# B&R Automation Studio project NAEUL004C00R13L518F00 (part 37)

### NtParam.typ - Change By Project
```iecst
(*2020-07-28*)

TYPE
	eNtParamAction :
		(
		NtParamActIdle,
		NtParamActCreateDir,
		NtParamActRead,
		NtParamActWrite,
		NtParamActLoad,
		NtParamActSave
		);
	tyNtParam : 	STRUCT
		tyDISettings : tyDigitalInputSettings := (diSafetyRlySig:=1,diEStopSig:=2,diCoverSWSig:=3,diUBAA:=4,diUBAB:=5,diUBAAStat:=6,diUBABStat:=7,diPusherExtRS:=12,diPusherRetRS:=13,diConvLftSen:=27,diConvMidSen:=28,diConvRgtSen:=29,diConvClrSen:=30,diOvenInfeedSigA:=0,diOvenInfeedSigB:=0,diLifterTimingBeltSen:=10,diLifterSafetyLmtSW1:=11,diLifterSafetyLmtSW2:=0,diMag1FixedClampRS:=0,diMag1FixedUnclampRS:=0,diMag1RemoteClampRS:=0,diMag1RemoteUnclampRS:=0,diMag2FixedClampRS:=0,diMag2FixedUnclampRS:=0,diMag2RemoteClampRS:=0,diMag2RemoteUnclampRS:=0,diMag3FixedClampRS:=0,diMag3FixedUnclampRS:=0,diMag3RemoteClampRS:=0,diMag3RemoteUnclampRS:=0,diInShutterOpenRS:=14,diInShutterCloseRS:=15,diOutShutterOpenRS:=16,diOutShutterCloseRS:=17,diMagPresentSen1:=8,diMagPresentSen2:=9,diMagPresentSen3:=0,diMagConvEntSen1:=0,diMagConvEntSen2:=0,diMagConvEntSen3:=0,diMag1AIVInPosSen1:=0,diMag1AIVInPosSen2:=0,diMag2AIVInPosSen1:=0,diMag2AIVInPosSen2:=0,diMag3AIVInPosSen1:=0,diMag3AIVInPosSen2:=0,diMag1OrientChkSen1:=0,diMag1OrientChkSen2:=0,diMag2OrientChkSen1:=0,diMag2OrientChkSen2:=0,diMag3OrientChkSen1:=0,diMag3OrientChkSen2:=0,diUSWidthChkSen:=0,diConvLineAInletSen:=0,diConvLineBInletSen:=0,diMagConvHeightSen1:=0,diMagConvHeightSen2:=0,diMagConvHeightSen3:=0,diMagConvSmallMagSen1:=0,diMagConvSmallMagSen2:=0,diMagConvSmallMagSen3:=0,diMagConvLargeMagSen1:=0,diMagConvLargeMagSen2:=0,diMagConvLargeMagSen3:=0,diMagConvCAB717MagSen1:=0,diMagConvCAB717MagSen2:=0,diMagConvCAB717MagSen3:=0,diMag1SelUnClampRS:=0,diMag2SelUnClampRS:=0,diMag3SelUnClampRS:=0,diMag1WallEngageRS:=0,diMag1WallDisengageRS:=0,diMag2WallEngageRS:=0,diMag2WallDisengageRS:=0,diMag3WallEngageRS:=0,diMag3WallDisengageRS:=0,diMag1SafetyBarExtRS:=0,diMag1SafetyBarRetRS:=0,diMag2SafetyBarExtRS:=0,diMag2SafetyBarRetRS:=0,diMag3SafetyBarExtRS:=0,diMag3SafetyBarRetRS:=0,diSOT1Receive:=0,diSOT1AIVError:=0,diSOT1AIVSizeLarge:=0,diSOT1AIVReady:=0,diSOT1AIVAvailable:=0,diSOT2Receive:=0,diSOT2AIVError:=0,diSOT2AIVSizeLarge:=0,diSOT2AIVReady:=0,diSOT2AIVAvailable:=0,diSOT3Receive:=0,diSOT3AIVError:=0,diSOT3AIVSizeLarge:=0,diSOT3AIVReady:=0,diSOT3AIVAvailable:=0,diSOT4Receive:=0,diSOT4AIVError:=0,diSOT4AIVSizeLarge:=0,diSOT4AIVReady:=0,diSOT4AIVAvailable:=0,diFleetManagerReady:=0,diPusherExtSlwSen:=0,diPusherRetSlwSen:=0,diMtrPshrTorqueSig:=0,diMtrPshrAlmSig:=0,diMagWidthChkSen:=0,diPshrAntiJam:=0,diInMagConvEntSen:=0,diInMagConvExtSen:=0,diInMagConvMidSen:=0,diOutMagConvEntSen:=0,diOutMagConvExtSen:=0,diOutMagConvMidSen:=0,diInMagConv2EntSen:=0,diInMagConv2ExtSen:=0,diInMagConv2MidSen:=0,diOutMagConv2EntSen:=0,diOutMagConv2ExtSen:=0,diOutMagConv2MidSen:=0,diLifterLmtSW:=0,diLifter2LmtSW:=0,diMtrOverloadSig:=0,diOutShutterOpenRS2:=0,diOutShutterCloseRS2:=0,diOutShutterOpenRS3:=0,diOutShutterCloseRS3:=0,diMag1FixedClampSen:=0,diMag2FixedClampSen:=0,diMag3FixedClampSen:=0,diCurtainSenPB:=0,diCurtainSen:=0,diCurtainSafetySig:=0,diHighMagDetSen1:=0,diHighMagDetSen2:=0,diHighMagDetSen3:=0,diInletStopperASen:=0,diScanComplSig:=0,diPCBScanSen:=0,diSPARE17:=0,diSPARE18:=0,diSPARE19:=0,diSPARE20:=0);
		tyDOSettings : tyDigitalOutputSettings := (diSafetyRlyRst:=1,diTLRed:=4,diTLAmber:=3,diTLGreen:=2,diBuzzer:=5,diUSBA:=8,diUSBB:=9,diOvenInfoSigA:=7,diOvenInfoSigB:=10,diPusherExtCtrl:=11,diStopperUnblkCtrlA:=0,diStopperUnblkCtrlB:=0,diMag1FixedClampCtrl:=0,diMag1RemoteClampCtrl:=0,diMag2FixedClampCtrl:=0,diMag2RemoteClampCtrl:=0,diMag3FixedClampCtrl:=0,diMag3RemoteClampCtrl:=0,diInShutterOpenCtrl:=15,diInShutterCloseCtrl:=16,diOutShutterOpenCtrl:=17,diOutShutterCloseCtrl:=18,diMag1ConvMtrIn:=0,diMag1ConvMtrOut:=0,diMag2ConvMtrIn:=0,diMag2ConvMtrOut:=0,diMag3ConvMtrIn:=0,diMag3ConvMtrOut:=0,diMag1SelClampCtrl:=0,diMag2SelClampCtrl:=0,diMag3SelClampCtrl:=0,diPushConvMtrOn:=12,diMag1WallEngageCtrl:=0,diMag2WallEngageCtrl:=0,diMag3WallEngageCtrl:=0,diMag1SafetyBarRetCtrl:=0,diMag2SafetyBarRetCtrl:=0,diMag3SafetyBarRetCtrl:=0,diSOT1MagError:=0,diSOT1MagSizeLarge:=0,diSOT1MagReady:=0,diSOT1MagAvailable:=0,diSOT2MagError:=0,diSOT2MagSizeLarge:=0,diSOT2MagReady:=0,diSOT2MagAvailable:=0,diSOT3MagError:=0,diSOT3MagSizeLarge:=0,diSOT3MagReady:=0,diSOT3MagAvailable:=0,diSOT4MagError:=0,diSOT4MagSizeLarge:=0,diSOT4MagReady:=0,diSOT4MagAvailable:=0,diMagAWOpenLimByp1:=0,diMagAWOpenLimByp2:=0,diMagAWOpenLimByp3:=0,diMagAWOpenLimByp4:=0,diMagAWSmallLimSen1:=0,diMagAWSmallLimSen2:=0,diMagAWSmallLimSen3:=0,diMagAWSmallLimSen4:=0,diMag1ReqToBring:=0,diMag1ReqToGet:=0,diMag2ReqToBring:=0,diMag2ReqToGet:=0,diMag3ReqToBring:=0,diMag3ReqToGet:=0,diMag4ReqToBring:=0,diMag4ReqToGet:=0,diMtrPshrExt:=0,diMtrPshrRet:=0,diMtrPshrOn:=0,diMtrPshrBrakeRls:=0,diMtrPshrSpdBinBit0:=0,diMtrPshrSpdBinBit1:=0,diMtrPshrSpdBinBit2:=0,diMtrPshrAlmRst:=0,diInMagConvMtrOn:=0,diOutMagConvMtrOn:=0,diInMagConv2MtrOn:=0,diOutMagConv2MtrOn:=0,diEntTopStprUnblkCtrl:=0,diMidTopStprUnblkCtrl:=0,diExtTopStprUnblkCtrl:=0,diMidBtmStprUnblkCtrl:=0,diExtBtmStprUnblkCtrl:=0,diEntTopStprUnblkCtrl2:=0,diMidTopStprUnblkCtrl2:=0,diExtTopStprUnblkCtrl2:=0,diMidBtmStprUnblkCtrl2:=0,diExtBtmStprUnblkCtrl2:=0,diMtrPwrRly:=0,diMag1FixedClampOpenCtrl:=0,diMag1RemoteClampOpenCtrl:=0,diMag2FixedClampOpenCtrl:=0,diMag2RemoteClampOpenCtrl:=0,diMag3FixedClampOpenCtrl:=0,diMag3RemoteClampOpenCtrl:=0,diOutShutterOpenCtrl2:=0,diOutShutterCloseCtrl2:=0,diOutShutterOpenCtrl3:=0,diOutShutterCloseCtrl3:=0,diBypCurtainSen:=0,diRstCurtainSen:=0,diBypCurtainPBLED:=6,diInletStopperRetCtrl:=0,diInletStopperExtCtrl:=0,diScanTrigSig:=0,diMag1ExitPCB:=0,diMag2ExitPCB:=0,diMag3ExitPCB:=0,diMag1SelUnClampCtrl:=0);
		bAWPusherPrep : BOOL := FALSE;
		bAWPrep : BOOL := TRUE;
		bLFPrep : BOOL := TRUE;
		bLeaderMc : BOOL := FALSE;
		bLFUsrSetPrep : BOOL := TRUE;
		diLFWidthLimit : DINT := 3000;
		bLFProdWidthChk : BOOL := FALSE;
		bUSWidthChkPrep : BOOL := FALSE;
		bLCSLFPrep : BOOL := TRUE;
		bLCSReqRcpPrep : BOOL := TRUE;
		bLCSManageRcpPrep : BOOL := TRUE;
		bLCSLiveDatPrep : BOOL := TRUE;
		bIPCSMEMA9851ExtdPrep : BOOL := TRUE;
		bVSMEMAPrep : BOOL := TRUE;
		bHermesPrep : BOOL := FALSE;
		bHermesRmtPrep : BOOL := FALSE;
		bOvenInfoPrep : BOOL := TRUE;
		bOvenInfoExtdPrep : BOOL := FALSE;
		bSSaverPrep : BOOL := TRUE;
		diAWPushPulOffsetInUM : DINT := 0;
		diWidthOffsetInUM : DINT := 0;
		sJobNo : STRING[30] := '2023-0529E01';
		usiNtAddr : USINT := 4;
		bProjLifterMagPlatform : BOOL := TRUE;
		bProjLaneBPrep : BOOL := FALSE;
		bProjBrdPerSltPrep : BOOL := FALSE;
		bProjLongBrdPrep : BOOL := FALSE;
		bProjInletShutPrep : BOOL := TRUE;
		bProjOutletShutPrep : BOOL := TRUE;
		bProjStopperAPrep : BOOL := FALSE;
		bProjStopperBPrep : BOOL := FALSE;
		bProjMag1ConvPrep : BOOL := FALSE;
		bProjMag2ConvPrep : BOOL := FALSE;
		bProjMag3ConvPrep : BOOL := FALSE;
		bProjLifter2Prep : BOOL := FALSE;
		bProjMagConvLane1Prep : BOOL := FALSE; (*TopBtm Conv, Lifter Conv*)
		bProjMagConvLane2Prep : BOOL := FALSE; (*TopBtm Conv, Lifter Conv*)
		bProjTopEntStprPrep : BOOL := FALSE; (*TopBtm Conv, Lifter Conv*)
		bProjTopMidStprPrep : BOOL := FALSE; (*TopBtm Conv, Lifter Conv*)
		bProjTopExtStprPrep : BOOL := FALSE; (*TopBtm Conv, Lifter Conv*)
		bProjBtmMidStprPrep : BOOL := FALSE; (*TopBtm Conv, Lifter Conv*)
		bProjBtmExtStprPrep : BOOL := FALSE; (*TopBtm Conv, Lifter Conv*)
		bProjTopEntStprPrep2 : BOOL := FALSE; (*TopBtm Conv, Lifter Conv*)
		bProjTopMidStprPrep2 : BOOL := FALSE; (*TopBtm Conv, Lifter Conv*)
		bProjTopExtStprPrep2 : BOOL := FALSE; (*TopBtm Conv, Lifter Conv*)
		bProjBtmMidStprPrep2 : BOOL := FALSE; (*TopBtm Conv, Lifter Conv*)
		bProjBtmExtStprPrep2 : BOOL := FALSE; (*TopBtm Conv, Lifter Conv*)
		bProjMagOrientChkSenPrep : BOOL := FALSE;
		bProjAGVPrep : BOOL := FALSE;
		bProjTCPAGVSigPrep : BOOL := FALSE;
		bProjBypsInitConvPrep : BOOL := TRUE;
		bProjRlsNewProdPrep : BOOL := FALSE;
		bProjBtnInsertRmvMag : BOOL := TRUE; (*fixed type*)
		bProjSOTSensorPrep : BOOL := FALSE;
		bProjMotorizedPusherPrep : BOOL := FALSE;
		bProjMagAWPrep : BOOL := FALSE;
		bProjMagSafetyBarPrep : BOOL := TRUE;
		diProjMagMinSlt : DINT := 1;
		diProjMagMaxSlt : DINT := 50;
		eProjMag : eULMag := ULMagTriple;
		eProjConvDir : eConvDir := ConvDirLToR;
		eProjMagConvDir : eConvDir := ConvDirLToL;
		eProjMagBuffferActLoad : eLifMagULUpdateData := BufferActLoadWhenStarted;
		eProjInMagConvDir : eConvDir := ConvDirRToL; (*Top*)
		eProjOutMagConvDir : eConvDir := ConvDirLToR; (*Bottom*)
		eProjLifterMagConvDir : eConvDir := ConvDirRToR; (*LifterConv*)
		eProjInMagConv2Dir : eConvDir := ConvDirRToL; (*Top*)
		eProjOutMagConv2Dir : eConvDir := ConvDirLToR; (*Bottom*)
		eProjLifterMagConv2Dir : eConvDir := ConvDirRToR; (*LifterConv*)
		sUsrFolderProgNm : STRING[15] := 'UsrFolder';
		sLibVersionProgNm : STRING[15] := 'LibVer';
		sTimeProgNm : STRING[15] := 'Time';
		sHWInfoProgNm : STRING[15] := 'HWInfo';
		sHWInfoDevice : STRING[3] := 'IF2';
		tyTLBuz : tyTLBuzIn1;
		sAlmProgNm : STRING[15] := 'Alarm';
		udiAlmFileKeepDay : UDINT := 30;
		sProdRcpProgNm : STRING[15] := 'ProdRcp';
		sProdRcpListFileNm : STRING[80] := 'ProductRecipeList.dat';
		sProdRcpSingleFileNm : STRING[80] := 'ProductRecipe.dat';
		sMpProdRcpProgNm : STRING[15] := 'MpProdRcp';
		sMpProdRcpFileNm : STRING[255] := 'MpProductRecipe.xml';
		sMpProdRcpPVNm : STRING[100] := 'MpProdRcp:a_tyMpProdRcp1';
		sMagRcpProgNm : STRING[15] := 'MagRcp';
		sMagRcpListFileNm : STRING[80] := 'MagazineRecipeList.dat';
		sMagRcpSingleFileNm : STRING[80] := 'MagazineRecipe.dat';
		sMcParamProgNm : STRING[15] := 'McParam';
		sMcParamFileNm : STRING[80] := 'MachineParameter.dat';
		sUsrMgmtProgNm : STRING[15] := 'UsrMgmt';
		sBffr1ProgNm : STRING[15] := 'Buffer 1';
		sBffr1FileNm : STRING[80] := 'Buffer1.dat';
		bBffr1NxtLoadSeq : BOOL := TRUE;
		sBffr2ProgNm : STRING[15] := 'Buffer 2';
		sBffr2FileNm : STRING[80] := 'Buffer2.dat';
		bBffr2NxtLoadSeq : BOOL := TRUE;
		sBffr3ProgNm : STRING[15] := 'Buffer 3';
		sBffr3FileNm : STRING[80] := 'Buffer3.dat';
		bBffr3NxtLoadSeq : BOOL := TRUE;
		sUSSMEMAAProgNm : STRING[15] := 'USSMEMA A';
		tUSSMEMAARstDlyTm : TIME := T#500ms;
		tUSSMEMAASigInChkTm : TIME := T#100ms;
		sUSSMEMABProgNm : STRING[15] := 'USSMEMA B';
		tUSSMEMABRstDlyTm : TIME := T#500ms;
		tUSSMEMABSigInChkTm : TIME := T#100ms;
		sUSSMEMA1ProgNm : STRING[15] := 'Mag1_US';
		tUSSMEMA1RstDlyTm : TIME := T#0s;
		tUSSMEMA1SigInChkTm : TIME := T#100ms;
		sUSSMEMA2ProgNm : STRING[15] := 'Mag2_US';
		tUSSMEMA2RstDlyTm : TIME := T#0s;
		tUSSMEMA2SigInChkTm : TIME := T#100ms;
		sUSSMEMA3ProgNm : STRING[15] := 'Mag3_US';
		tUSSMEMA3RstDlyTm : TIME := T#0s;
		tUSSMEMA3SigInChkTm : TIME := T#100ms;
		sDSSMEMA1ProgNm : STRING[15] := 'Mag1_DS';
		tDSSMEMA1RstDlyTm : TIME := T#0s;
		tDSSMEMA1SigInChkTm : TIME := T#100ms;
		sDSSMEMA2ProgNm : STRING[15] := 'Mag2_DS';
		tDSSMEMA2RstDlyTm : TIME := T#0s;
		tDSSMEMA2SigInChkTm : TIME := T#100ms;
		sDSSMEMA3ProgNm : STRING[15] := 'Mag3_DS';
		tDSSMEMA3RstDlyTm : TIME := T#0s;
		tDSSMEMA3SigInChkTm : TIME := T#100ms;
		sInShutterProgNm : STRING[15] := 'Inlet Shutter';
		bInShutterTwoCtrlIn : BOOL := TRUE;
		tInShutterExtTO : TIME := T#20s;
		tInShutterRetTO : TIME := T#20s;
		sOutShutterProgNm : STRING[15] := 'Outlet Shutter';
		bOutShutterTwoCtrlIn : BOOL := TRUE;
		tOutShutterExtTO : TIME := T#20s;
		tOutShutterRetTO : TIME := T#20s;
		sSelClamp1ProgNm : STRING[15] := 'Sel Clamp 1';
		bSelClamp1TwoCtrlIn : BOOL := TRUE;
		tSelClamp1ExtDlyTm : TIME := T#10s;
		tSelClamp1RetDlyTm : TIME := T#10s;
		sSelClamp2ProgNm : STRING[15] := 'Sel Clamp 2';
		bSelClamp2TwoCtrlIn : BOOL := FALSE;
		tSelClamp2ExtDlyTm : TIME := T#10s;
		tSelClamp2RetDlyTm : TIME := T#10s;
		sSelClamp3ProgNm : STRING[15] := 'Sel Clamp 3';
		bSelClamp3TwoCtrlIn : BOOL := FALSE;
		tSelClamp3ExtDlyTm : TIME := T#10s;
		tSelClamp3RetDlyTm : TIME := T#10s;
		sTopEntStprProgNm : STRING[15] := 'Top Ent Stpr';
		bTopEntStprTwoCtrlIn : BOOL := FALSE;
		tTopEntStprExtDlyTm : TIME := T#1s;
		tTopEntStprRetDlyTm : TIME := T#1s;
		sTopMidStprProgNm : STRING[15] := 'Top Mid Stpr';
		bTopMidStprTwoCtrlIn : BOOL := FALSE;
		tTopMidStprExtDlyTm : TIME := T#1s;
		tTopMidStprRetDlyTm : TIME := T#1s;
		sTopExtStprProgNm : STRING[15] := 'Top Ext Stpr';
		bTopExtStprTwoCtrlIn : BOOL := FALSE;
		tTopExtStprExtDlyTm : TIME := T#1s;
		tTopExtStprRetDlyTm : TIME := T#1s;
		sBtmMidStprProgNm : STRING[15] := 'Top Mid Stpr';
		bBtmMidStprTwoCtrlIn : BOOL := FALSE;
		tBtmMidStprExtDlyTm : TIME := T#1s;
		tBtmMidStprRetDlyTm : TIME := T#1s;
		sBtmExtStprProgNm : STRING[15] := 'Btm Ext Stpr';
		bBtmExtStprTwoCtrlIn : BOOL := FALSE;
		tBtmExtStprExtDlyTm : TIME := T#1s;
		tBtmExtStprRetDlyTm : TIME := T#1s;
		sTopEntStprProgNm2 : STRING[15] := 'Top Ent Stpr2';
		bTopEntStprTwoCtrlIn2 : BOOL := FALSE;
		tTopEntStprExtDlyTm2 : TIME := T#1s;
		tTopEntStprRetDlyTm2 : TIME := T#1s;
		sTopMidStprProgNm2 : STRING[15] := 'Top Mid Stpr2';
		bTopMidStprTwoCtrlIn2 : BOOL := FALSE;
		tTopMidStprExtDlyTm2 : TIME := T#1s;
		tTopMidStprRetDlyTm2 : TIME := T#1s;
		sTopExtStprProgNm2 : STRING[15] := 'Top Ext Stpr2';
		bTopExtStprTwoCtrlIn2 : BOOL := FALSE;
		tTopExtStprExtDlyTm2 : TIME := T#1s;
		tTopExtStprRetDlyTm2 : TIME := T#1s;
		sBtmMidStprProgNm2 : STRING[15] := 'Top Mid Stpr2';
		bBtmMidStprTwoCtrlIn2 : BOOL := FALSE;
		tBtmMidStprExtDlyTm2 : TIME := T#1s;
		tBtmMidStprRetDlyTm2 : TIME := T#1s;
		sBtmExtStprProgNm2 : STRING[15] := 'Btm Ext Stpr2';
		bBtmExtStprTwoCtrlIn2 : BOOL := FALSE;
		tBtmExtStprExtDlyTm2 : TIME := T#1s;
		tBtmExtStprRetDlyTm2 : TIME := T#1s;
		sStopperAProgNm : STRING[15] := 'Stopper A';
		bStopperATwoCtrlIn : BOOL := FALSE;
		tStopperAExtDlyTm : TIME := T#1s;
		tStopperARetDlyTm : TIME := T#1s;
		sStopperBProgNm : STRING[15] := 'Stopper B';
		bStopperBTwoCtrlIn : BOOL := FALSE;
		tStopperBExtDlyTm : TIME := T#1s;
		tStopperBRetDlyTm : TIME := T#1s;
		sPshrConvProgNm : STRING[15] := 'PusherConv';
		bPshrConvOnDirMod : BOOL := FALSE;
		tPshrConvMtrOffDlyTm : TIME := T#0s;
		tPshrConvPshrExtTO : TIME := T#20s;
		tPshrConvPshrRetTO : TIME := T#20s;
		sMag1SafetyBarProgNm : STRING[15] := 'Mag1 SafetyBar';
		bMag1SafetyBarTwoCtrlIn : BOOL := FALSE;
		tMag1SafetyBarExtTO : TIME := T#20s;
		tMag1SafetyBarRetTO : TIME := T#20s;
		sMag2SafetyBarProgNm : STRING[15] := 'Mag2 SafetyBar';
		bMag2SafetyBarTwoCtrlIn : BOOL := FALSE;
		tMag2SafetyBarExtTO : TIME := T#20s;
		tMag2SafetyBarRetTO : TIME := T#20s;
		sMag3SafetyBarProgNm : STRING[15] := 'Mag3 SafetyBar';
		bMag3SafetyBarTwoCtrlIn : BOOL := FALSE;
		tMag3SafetyBarExtTO : TIME := T#20s;
		tMag3SafetyBarRetTO : TIME := T#20s;
		sMag1AWEngageProgNm : STRING[15] := 'Mag1 AWEngage';
		bMag1AWEngageTwoCtrlIn : BOOL := FALSE;
		tMag1AWEngageExtTO : TIME := T#20s;
		tMag1AWEngageRetTO : TIME := T#20s;
		sMag2AWEngageProgNm : STRING[15] := 'Mag2 AWEngage';
		bMag2AWEngageTwoCtrlIn : BOOL := FALSE;
		tMag2AWEngageExtTO : TIME := T#20s;
		tMag2AWEngageRetTO : TIME := T#20s;
		sMag3AWEngageProgNm : STRING[15] := 'Mag3 AWEngage';
		bMag3AWEngageTwoCtrlIn : BOOL := FALSE;
		tMag3AWEngageExtTO : TIME := T#20s;
		tMag3AWEngageRetTO : TIME := T#20s;
		sMagConv1ProgNm : STRING[15] := 'MagConv 1';
		bMagConv1OnDirMod : BOOL := FALSE;
		tMagConv1MtrOffDlyTm : TIME := T#0s;
		tMagConv1ClprClampTO : TIME := T#20s;
		tMagConv1ClprUnclampTO : TIME := T#20s;
		sMagConv2ProgNm : STRING[15] := 'MagConv 2';
		bMagConv2OnDirMod : BOOL := FALSE;
		tMagConv2MtrOffDlyTm : TIME := T#0s;
		tMagConv2ClprClampTO : TIME := T#20s;
		tMagConv2ClprUnclampTO : TIME := T#20s;
		sMagConv3ProgNm : STRING[15] := 'MagConv 3';
		bMagConv3OnDirMod : BOOL := FALSE;
		tMagConv3MtrOffDlyTm : TIME := T#0s;
		tMagConv3ClprClampTO : TIME := T#20s;
		tMagConv3ClprUnclampTO : TIME := T#20s;
		sMtrPshrProgNm : STRING[15] := 'Motorized Pshr';
		bMtrPshrDir : BOOL := TRUE;
		tMtrPshrAlmRstTm : TIME := T#1s;
		tMtrPshrAlmTrigTm : TIME := T#1s;
		tMtrPshrExtTO : TIME := T#20s;
		tMtrPshrRetTO : TIME := T#20s;
		diMtrPshrExtSlowSpd : DINT := 1;
		diMtrPshrRetSlowSpd : DINT := 3;
		diMtrPshrExtNomSpd : DINT := 4;
		diMtrPshrRetNomSpd : DINT := 8;
		diMtrPshrExtTorq : DINT := 50;
		diMtrPshrRetTorq : DINT := 100;
		diMtrPshrStartTorq : DINT := 100;
		sInMagConvProgNm : STRING[15] := 'Input Mag Conv'; (*Top*)
		bInMagConvOnDirMod : BOOL := FALSE;
		tInMagConvMtrOffDlyTm : TIME := T#500ms;
		sOutMagConvProgNm : STRING[15] := 'Output Mag Conv'; (*Bottom*)
		bOutMagConvOnDirMod : BOOL := FALSE;
		tOutMagConvMtrOffDlyTm : TIME := T#100ms;
		sLifterMagProgNm : STRING[15] := 'Lifter Mag Conv'; (*Lifter*)
		bLifterMagOnDirMod : BOOL := FALSE;
		tLifterMagMtrOffDlyTm : TIME := T#2s;
		tLifterMagClprClampTO : TIME := T#20s;
		tLifterMagClprUnclampTO : TIME := T#20s;
		sInMagConv2ProgNm : STRING[15] := 'In Mag Conv2';
		bInMagConv2OnDirMod : BOOL := FALSE;
		tInMagConv2MtrOffDlyTm : TIME := T#500ms;
		sOutMagConv2ProgNm : STRING[15] := 'Out Mag Conv2';
		bOutMagConv2OnDirMod : BOOL := FALSE;
		tOutMagConv2MtrOffDlyTm : TIME := T#100ms;
		sLifterMag2ProgNm : STRING[15] := 'Lift Mag Conv2';
		bLifterMag2OnDirMod : BOOL := FALSE;
		tLifterMag2MtrOffDlyTm : TIME := T#2s;
		tLifterMagClprClampTO2 : TIME := T#20s;
		tLifterMagClprUnclampTO2 : TIME := T#20s;
		sAWPushPullProgNm : STRING[15] := 'AWPusher';
		sAWPushPullDevice : STRING[3] := 'IF7';
		usiAWPushPullNode : USINT := 22;
		bAWPushPullDir : BOOL := FALSE;
		bAWPushPullDirBl : BOOL := FALSE;
		diAWPushPullPitchInUM : DINT := 3000;
		diAWPushPullMovBlDistInUM : DINT := 3000;
		tyAWPushPullParamInHm : tyMotionCANParamInHm := (diStartVelInUMPS:=15000,diAcc:=50);
		tyAWPushPullParamInConvert : tyMotionCANParamInConvert := (diPitchInUM:=3000);
		tyAWPushPullParam : tyMotionParam := (diAccInMS:=500,diDecInMS:=500,diAutoSpdInUMPS:=15000);
		tyAWPushPullTuning : tyMotionCANTuning := (diAsdaA2Inertia:=76,diAsdaA2PosLoopGain:=53,diAsdaA2PosFFGain:=50,diAsdaA2SpdLoopGain:=213,diAsdaA2SpdIntegral:=34,diAsdaA2LowPassFltr:=49,diAsdaA2AntiInterGain:=34,diAsdaA2FirstTorqueCmd:=300,diLex28LTNDderivativeGain_P800:=0,diLex28LTNIintegralGain_P801:=0,diLex28LTNIVdeIntlGain_P802:=0,diLex28LTNPpropotionalGain_P803:=0,diLex28LTNUSERGAIN_P804:=0,diLex28NLAFFLPFHZspringFil_P805:=0,diLex28NLFILTDAMPING_P814:=0,diLex28NLFILTT1_P815:=0,diPronetInertia:=100,diPronetRealTimeAutoAdjSet:=0,diPronetPosLoopGain:=40,diPronetSpdLoopGain:=250,diPronetSpdIntegral:=200,diPronetTorqueFilter:=100,diPronetPosFeedForward:=0,diPronetLowSpeedTestFiltering:=10,diPronetStopMode:=5);
		eAWPushPullServoMotorType : eServoMotorType := DeltaAsdaA2; (*Selection of  Motor Brand*)
		sAWProgNm : STRING[15] := 'AWOpen';
		sAWDevice : STRING[3] := 'IF7';
		usiAWNode : USINT := 16;
		bAWDir : BOOL := TRUE;
		bAWDirBl : BOOL := FALSE;
		diAWPitchInUM : DINT := 3000;
		diAWMovBlDistInUM : DINT := 3000;
		tyAWParamInHm : tyMotionCANParamInHm := (diStartVelInUMPS:=15000,diAcc:=25);
		tyAWParamInConvert : tyMotionCANParamInConvert := (diPitchInUM:=3000);
		tyAWParam : tyMotionParam := (diAccInMS:=500,diDecInMS:=500,diAutoSpdInUMPS:=15000);
		tyAWTuning : tyMotionCANTuning := (diAsdaA2Inertia:=76,diAsdaA2PosLoopGain:=53,diAsdaA2PosFFGain:=50,diAsdaA2SpdLoopGain:=213,diAsdaA2SpdIntegral:=34,diAsdaA2LowPassFltr:=49,diAsdaA2AntiInterGain:=34,diAsdaA2FirstTorqueCmd:=300,diLex28LTNDderivativeGain_P800:=0,diLex28LTNIintegralGain_P801:=0,diLex28LTNIVdeIntlGain_P802:=0,diLex28LTNPpropotionalGain_P803:=0,diLex28LTNUSERGAIN_P804:=0,diLex28NLAFFLPFHZspringFil_P805:=0,diLex28NLFILTDAMPING_P814:=0,diLex28NLFILTT1_P815:=0,diPronetInertia:=0,diPronetRealTimeAutoAdjSet:=0,diPronetPosLoopGain:=80,diPronetSpdLoopGain:=750,diPronetSpdIntegral:=600,diPronetTorqueFilter:=4,diPronetPosFeedForward:=0,diPronetLowSpeedTestFiltering:=0,diPronetStopMode:=5);
		eAWServoMotorType : eServoMotorType := DeltaAsdaA2; (*Selection of  Motor Brand*)
		sTravProgNm : STRING[15] := 'Trav';
		sTravDevice : STRING[3] := 'IF7';
		usiTravNode : USINT := 18;
		bTravDir : BOOL := TRUE;
		tyTravParamInHm : tyMotionCANParamInHm := (diStartVelInUMPS:=50000,diAcc:=25);
		tyTravParamInConvert : tyMotionCANParamInConvert := (diPitchInUM:=25000,diPrimaryGearRatio:=1,diSecondaryGearRatio:=1); (*belt190530,estun1048576*)
		tyTravParam : tyMotionParam := (diAccInMS:=300,diDecInMS:=300,diAutoSpdInUMPS:=100000); (*500;1500*)
		tyTravTuning : tyMotionCANTuning := (diAsdaA2Inertia:=76,diAsdaA2PosLoopGain:=53,diAsdaA2PosFFGain:=50,diAsdaA2SpdLoopGain:=213,diAsdaA2SpdIntegral:=34,diAsdaA2LowPassFltr:=49,diAsdaA2AntiInterGain:=34,diAsdaA2FirstTorqueCmd:=300,diLex28LTNDderivativeGain_P800:=0,diLex28LTNIintegralGain_P801:=0,diLex28LTNIVdeIntlGain_P802:=0,diLex28LTNPpropotionalGain_P803:=0,diLex28LTNUSERGAIN_P804:=0,diLex28NLAFFLPFHZspringFil_P805:=0,diLex28NLFILTDAMPING_P814:=0,diLex28NLFILTT1_P815:=0,diPronetInertia:=0,diPronetRealTimeAutoAdjSet:=0,diPronetPosLoopGain:=80,diPronetSpdLoopGain:=750,diPronetSpdIntegral:=600,diPronetTorqueFilter:=4,diPronetPosFeedForward:=0,diPronetLowSpeedTestFiltering:=0,diPronetStopMode:=5);
		eTravServoMotorType : eServoMotorType := DeltaAsdaA2; (*Selection of  Motor Brand*)
		diTravAutoSpdLongBrdInUMPS : DINT := 100000;
		sLifterProgNm : STRING[15] := 'LifterBtm';
		sLifterDevice : STRING[3] := 'IF7';
		usiLifterNode : USINT := 17;
		bLifterDir : BOOL := TRUE;
		tyLifterParamInHm : tyMotionCANParamInHm := (diStartVelInUMPS:=25000,diAcc:=25);
		tyLifterParamInConvert : tyMotionCANParamInConvert := (diPitchInUM:=10000,diPrimaryGearRatio:=1,diSecondaryGearRatio:=1); (*estun1048576*)
		tyLifterParam : tyMotionParam := (diAccInMS:=300,diDecInMS:=300,diAutoSpdInUMPS:=50000); (*closed spd150, 10s spd 5000(000)*)
		tyLifterTuning : tyMotionCANTuning := (diAsdaA2Inertia:=62,diAsdaA2PosLoopGain:=64,diAsdaA2PosFFGain:=50,diAsdaA2SpdLoopGain:=257,diAsdaA2SpdIntegral:=41,diAsdaA2LowPassFltr:=40,diAsdaA2AntiInterGain:=41,diAsdaA2FirstTorqueCmd:=300,diLex28LTNDderivativeGain_P800:=1116,diLex28LTNIintegralGain_P801:=321,diLex28LTNIVdeIntlGain_P802:=319,diLex28LTNPpropotionalGain_P803:=482,diLex28LTNUSERGAIN_P804:=1000,diLex28NLAFFLPFHZspringFil_P805:=5000,diLex28NLFILTDAMPING_P814:=35,diLex28NLFILTT1_P815:=25,diPronetInertia:=0,diPronetRealTimeAutoAdjSet:=0,diPronetPosLoopGain:=40,diPronetSpdLoopGain:=250,diPronetSpdIntegral:=500,diPronetTorqueFilter:=100,diPronetPosFeedForward:=0,diPronetLowSpeedTestFiltering:=10,diPronetStopMode:=5);
		eLifterServoMotorType : eServoMotorType := DeltaAsdaA2; (*Selection of  Motor Brand*)
		sLifterProgNm2 : STRING[15] := 'Lifter2';
		sLifterDevice2 : STRING[3] := 'IF7';
		usiLifterNode2 : USINT := 25;
		bLifterDir2 : BOOL := TRUE;
		tyLifterParamInHm2 : tyMotionCANParamInHm := (diStartVelInUMPS:=25000,diAcc:=25);
		tyLifterParamInConvert2 : tyMotionCANParamInConvert := (diPitchInUM:=10000,diPulsePerRev:=1048576); (*estun1048576*)
		tyLifterParam2 : tyMotionParam := (diAccInMS:=500,diDecInMS:=500,diAutoSpdInUMPS:=50000); (*closed spd150*)
		tyLifterTuning2 : tyMotionCANTuning := (diAsdaA2Inertia:=62,diAsdaA2PosLoopGain:=64,diAsdaA2PosFFGain:=50,diAsdaA2SpdLoopGain:=257,diAsdaA2SpdIntegral:=41,diAsdaA2LowPassFltr:=40,diAsdaA2AntiInterGain:=41,diAsdaA2FirstTorqueCmd:=300,diLex28LTNDderivativeGain_P800:=1116,diLex28LTNIintegralGain_P801:=321,diLex28LTNIVdeIntlGain_P802:=319,diLex28LTNPpropotionalGain_P803:=482,diLex28LTNUSERGAIN_P804:=1000,diLex28NLAFFLPFHZspringFil_P805:=5000,diLex28NLFILTDAMPING_P814:=35,diLex28NLFILTT1_P815:=25,diPronetInertia:=0,diPronetRealTimeAutoAdjSet:=0,diPronetPosLoopGain:=40,diPronetSpdLoopGain:=250,diPronetSpdIntegral:=500,diPronetTorqueFilter:=100,diPronetPosFeedForward:=0,diPronetLowSpeedTestFiltering:=10,diPronetStopMode:=5);
		eLifterServoMotorType2 : eServoMotorType := DeltaAsdaA2; (*Selection of  Motor Brand*)
		sDIProgNm : STRING[15] := 'DInput';
		sAGVProgNm : STRING[15] := 'AGV';
		sAGVMag1ProgNm : STRING[15] := 'AGVMag 1';
		sAGVMag2ProgNm : STRING[15] := 'AGVMag 2';
		sAGVMag3ProgNm : STRING[15] := 'AGVMag 3';
		sHermesProgNm : STRING[15] := 'Hermes';
		sHermesRetainFileNm : STRING[80] := 'Hermes.dat';
		sHermesConfigFileNm : STRING[80] := 'Hermes.dat';
		sUSHermesAProgNm : STRING[15] := 'USHermes A';
		udiUSHermesAFileKeepDay : UDINT := 7;
		udiUSHermesAAliveTmInSec : UDINT := 5;
		tUSHermesAConnTO : TIME := T#30s;
		sUSHermesBProgNm : STRING[15] := 'USHermes B';
		udiUSHermesBFileKeepDay : UDINT := 7;
		udiUSHermesBAliveTmInSec : UDINT := 5;
		tUSHermesBConnTO : TIME := T#30s;
		sRmtHermesProgNm : STRING[15] := 'RmtHermes';
		sRmtHermesConfigFileNm : STRING[80] := 'RmtHermes.dat';
		udiRmtHermesFileKeepDay : UDINT := 7;
		udiRmtHermesAliveTmInSec : UDINT := 5;
		udiRmtHermesSndBffrSize : UDINT := 65536;
		udiRmtHermesRcvBffrSize : UDINT := 65536;
		sLFLeaderProgNm : STRING[15] := 'LFLeader';
		tLFLeaderOnlineChkDlyTm : TIME := T#20s;
		tLFLeaderSetTmOffDlyTm : TIME := T#10s;
		sLFFollowerProgNm : STRING[15] := 'Follower';
		sFollower1ProgNm : STRING[15] := 'Follower 1';
		sFollower2ProgNm : STRING[15] := 'Follower 2';
		sLCSProgNm : STRING[15] := 'LCS';
		sLCSMngRcpProgNm : STRING[15] := 'LCSMngRcp';
		sLCSLFProgNm : STRING[15] := 'LCSLF';
		sOpsTravLifULProgNm : STRING[15] := 'OpsTravLifUL';
		sOpsMagUL1ProgNm : STRING[15] := 'OpsMagUL 1';
		sOpsMagUL2ProgNm : STRING[15] := 'OpsMagUL 2';
		sOpsMagUL3ProgNm : STRING[15] := 'OpsMagUL 3';
		sOpsMagConvUL1ProgNm : STRING[15] := 'OpsMagConvUL 1';
		sOpsMagConvUL2ProgNm : STRING[15] := 'OpsMagConvUL 2';
		sOpsMagConvUL3ProgNm : STRING[15] := 'OpsMagConvUL 3';
		sOpsInMagConv : STRING[15] := 'In Mag Conv';
		sOpsOutMagConv : STRING[15] := 'Out Mag Conv';
		sOpsMagConvStprProgNm : STRING[15] := 'OpsMagConvStpr1';
		sOpsMagConvStprProgNm1 : STRING[15] := 'OpsMagConvStpr2';
		tyProdRcpWidth : tyUILmt := (diMax:=460000,diMin:=70000);
		tyProdRcpMinSlt : tyUILmt := (diMax:=50,diMin:=1);
		tyProdRcpMaxSlt : tyUILmt := (diMax:=50,diMin:=1);
		tyProdRcpPitch : tyUILmt := (diMax:=49,diMin:=1);
		tyProdRcpBrdPerSlt : tyUILmt := (diMax:=2,diMin:=1);
		tyProdRcpMcModA : tyUILmt := (diMax:=2,diMin:=0);
		tyProdRcpMcModAB : tyUILmt := (diMax:=8,diMin:=0);
		tyProdRcpOvenMinReqFreeBffr : tyUILmt := (diMax:=50,diMin:=0);
		tyUISSaverTm : tyUILmt := (diMax:=1800,diMin:=10);
		tyUIConvInitTm : tyUILmt := (diMax:=60000,diMin:=3000);
		tyUIMagConvRunTm : tyUILmt := (diMax:=60000,diMin:=5000);
		tyUILifterTopPos : tyUILmt := (diMax:=750000,diMin:=-10000);
		tyUILifterBtmPos : tyUILmt := (diMax:=750000,diMin:=-10000);
		tyUITranInErrDlyTm : tyUILmt := (diMax:=120000,diMin:=1000);
		tyUIOvenMaxBffrBtwnMc : tyUILmt := (diMax:=100,diMin:=1);
		tyUIHermesSndAliveTm : tyUILmt := (diMax:=1800000,diMin:=5000);
		tyUIHermesLnID : tyUILmt := (diMax:=1000,diMin:=1);
		tyUIAntiGapSenOnTm : tyUILmt := (diMax:=5000,diMin:=0);
		tyUIAntiGapSenOffTm : tyUILmt := (diMax:=5000,diMin:=0);
		tyUISltToSltDist : tyUILmt := (diMax:=50000,diMin:=1000);
		tyUIAWTargetPos : tyUILmt := (diMax:=250000,diMin:=100000);
		tyUIAWStepSize : tyUILmt := (diMax:=400000,diMin:=-400000);
		tyUIAWNomSpd : tyUILmt := (diMax:=15000,diMin:=5000);
		tyUIAWSlwSpd : tyUILmt := (diMax:=15000,diMin:=5000);
		tyUITravTargetPos : tyUILmt := (diMax:=1170000,diMin:=-20000);
		tyUITravStepSize : tyUILmt := (diMax:=1170000,diMin:=-1170000);
		tyUITravNomSpd : tyUILmt := (diMax:=100000,diMin:=5000);
		tyUITravSlwSpd : tyUILmt := (diMax:=100000,diMin:=5000);
		tyUILifterTargetPos : tyUILmt := (diMax:=750000,diMin:=0);
		tyUILifterStepSize : tyUILmt := (diMax:=750000,diMin:=-750000);
		tyUILifterNomSpd : tyUILmt := (diMax:=100000,diMin:=5000);
		tyUILifterSlwSpd : tyUILmt := (diMax:=100000,diMin:=5000);
		tyUIMagAWTargetPos : tyUILmt := (diMax:=250000,diMin:=70000);
		tyUIMagAWStepSize : tyUILmt := (diMax:=250000,diMin:=-250000);
		tyUIMagAWNomSpd : tyUILmt := (diMax:=15000,diMin:=1000);
		tyUIMagAWSlwSpd : tyUILmt := (diMax:=15000,diMin:=1000);
		tyUILFIndexBeforeOven : tyUILmt := (diMax:=100,diMin:=1);
		tyUILFIndexAfterOven : tyUILmt := (diMax:=100,diMin:=1);
		sUIDefaultLoginNm : STRING[30];
		sUIDefaultLoginPw : STRING[30];
		tShutterWaitTmr : TIME := T#500ms;
		tyUIAWOffset : tyUILmt := (diMax:=2000,diMin:=-2000);
		bAutoLogoutPrep : BOOL := TRUE;
		tyUIAutoLogoutTm : tyUILmt := (diMax:=1800000,diMin:=60000);
		bMagAutoVerifyPrep : BOOL := FALSE;
		tyUIMcParamMagAutoEntSenTm : tyUILmt := (diMax:=5000,diMin:=0);
		bProjAIVInPosSenPrep : BOOL := FALSE;
		sMpNtParamFileNm : STRING[255] := 'NutekParameter.xml';
		sMpNtParamPVNm : STRING[100] := 'NtParam:tyMpNtParamCurr1';
		tyNetworkMode : tyUILmt := (diMax:=1,diMin:=0);
		bHermesSvyPrep : BOOL := FALSE; (*Supervisory Hermes Preparation*)
		bHermesSvyFirstMcInTheLine1 : BOOL := FALSE; (*Turn On this for Loader / Destacker Only. Other type of machine turns off.*)
		bHermesSvyMagTypeMc : BOOL := FALSE; (*Turn On this for Loader (Magazine type machine) Only. Other type of machine turns off.
*)
		sSvyHermesProgNm : STRING[15] := 'SvyHermes';
		sSvyHermesConfigFileNm : STRING[80] := 'SvyHermes.dat';
		udiSvyHermesFileKeepDay : UDINT := 7;
		udiSvyHermesAliveTmInSec : UDINT := 5;
		tSvyHermesConnTO : TIME := T#30s;
		sSvyHermesRetainFileNm : STRING[80] := 'WorkOrder.dat';
		sDSHermesRetainFileNm : STRING[80] := 'BoardData.dat';
		rMachineCycleTime : REAL := 6.0; (*1.0 = 1 second*)
		rAutoWidthCycleTime : REAL := 30.0; (*30.0 = 30 seconds*)
		bHermesScannerPrep1 : BOOL := FALSE; (*Turn On if machine has fixed scanner or handheld scanner*)
		iInput : INT := 1; (*Total Inlet, Single Track = 1, Dual Track = 2, and so on*)
		iOutput : INT := 1; (*Total Outlet, Single Track = 1, Dual Track = 2, and so on*)
		bLFProdWidth2Prep : BOOL := FALSE;
		tLFFollowerOnlineChkDlyTm : TIME := T#30s;
		sMagAW1ProgNm : STRING[15] := 'MagAWOpen1';
		sMagAW1Device : STRING[3] := 'IF7';
		usiMagAW1Node : USINT := 19;
		bMagAW1Dir : BOOL := TRUE;
		bMagAW1DirBl : BOOL := FALSE;
		diMagAW1PitchInUM : DINT := 10000;
		diMagAW1MovBlDistInUM : DINT := 0;
		tyMagAW1ParamInHm : tyMotionCANParamInHm := (diStartVelInUMPS:=10000,diAcc:=25);
		tyMagAW1ParamInConvert : tyMotionCANParamInConvert := (diPitchInUM:=10000);
		tyMagAW1Param : tyMotionParam := (diAccInMS:=500,diDecInMS:=500,diAutoSpdInUMPS:=20000);
		tyMagAW1Tuning : tyMotionCANTuning := (diAsdaA2Inertia:=14,diAsdaA2PosLoopGain:=150,diAsdaA2PosFFGain:=50,diAsdaA2SpdLoopGain:=200,diAsdaA2SpdIntegral:=124,diAsdaA2LowPassFltr:=13,diAsdaA2AntiInterGain:=124,diAsdaA2FirstTorqueCmd:=300);
		diMagAW1EngageSpdInUMPS : DINT := 5000;
		eMagAW1ServoMotorType : eServoMotorType := DeltaAsdaA2; (*Selection of  Motor Brand*)
		diMag1WidthOffsetInUM : DINT := 0;
		sMagAW2ProgNm : STRING[15] := 'MagAWOpen2';
		sMagAW2Device : STRING[3] := 'IF7';
		usiMagAW2Node : USINT := 20;
		bMagAW2Dir : BOOL := TRUE;
		bMagAW2DirBl : BOOL := FALSE;
		diMagAW2PitchInUM : DINT := 10000;
		diMagAW2MovBlDistInUM : DINT := 0;
		tyMagAW2ParamInHm : tyMotionCANParamInHm := (diStartVelInUMPS:=10000,diAcc:=25);
		tyMagAW2ParamInConvert : tyMotionCANParamInConvert := (diPitchInUM:=10000);
		tyMagAW2Param : tyMotionParam := (diAccInMS:=500,diDecInMS:=500,diAutoSpdInUMPS:=20000);
		tyMagAW2Tuning : tyMotionCANTuning := (diAsdaA2Inertia:=14,diAsdaA2PosLoopGain:=150,diAsdaA2PosFFGain:=50,diAsdaA2SpdLoopGain:=200,diAsdaA2SpdIntegral:=124,diAsdaA2LowPassFltr:=13,diAsdaA2AntiInterGain:=124,diAsdaA2FirstTorqueCmd:=300);
		diMagAW2EngageSpdInUMPS : DINT := 5000;
		eMagAW2ServoMotorType : eServoMotorType := DeltaAsdaA2; (*Selection of  Motor Brand*)
		diMag2WidthOffsetInUM : DINT := 0;
		sMagAW3ProgNm : STRING[15] := 'MagAWOpen3';
		sMagAW3Device : STRING[3] := 'IF7';
		usiMagAW3Node : USINT := 21;
		bMagAW3Dir : BOOL := TRUE;
		bMagAW3DirBl : BOOL := FALSE;
		diMagAW3PitchInUM : DINT := 10000;
		diMagAW3MovBlDistInUM : DINT := 0;
		tyMagAW3ParamInHm : tyMotionCANParamInHm := (diStartVelInUMPS:=10000,diAcc:=25);
		tyMagAW3ParamInConvert : tyMotionCANParamInConvert := (diPitchInUM:=10000);
		tyMagAW3Param : tyMotionParam := (diAccInMS:=500,diDecInMS:=500,diAutoSpdInUMPS:=20000);
		tyMagAW3Tuning : tyMotionCANTuning := (diAsdaA2Inertia:=14,diAsdaA2PosLoopGain:=150,diAsdaA2PosFFGain:=50,diAsdaA2SpdLoopGain:=200,diAsdaA2SpdIntegral:=124,diAsdaA2LowPassFltr:=13,diAsdaA2AntiInterGain:=124,diAsdaA2FirstTorqueCmd:=300);
		diMagAW3EngageSpdInUMPS : DINT := 5000;
		eMagAW3ServoMotorType : eServoMotorType := DeltaAsdaA2; (*Selection of  Motor Brand*)
		diMag3WidthOffsetInUM : DINT := 0;
		sMachineProgNm : STRING[15] := 'Machine';
		sUSSOT1ProgNm : STRING[15] := 'USSOT1';
		tUSSOT1RstDlyTm : TIME := T#0s;
		tUSSOT1SigInChkTm : TIME := T#100ms;
		sUSSOT2ProgNm : STRING[15] := 'USSOT2';
		tUSSOT2RstDlyTm : TIME := T#0s;
		tUSSOT2SigInChkTm : TIME := T#100ms;
		sUSSOT3ProgNm : STRING[15] := 'USSOT3';
		tUSSOT3RstDlyTm : TIME := T#0s;
		tUSSOT3SigInChkTm : TIME := T#100ms;
		sDSSOT1ProgNm : STRING[15] := 'DSSOT1';
		tDSSOT1RstDlyTm : TIME := T#0s;
		tDSSOT1SigInChkTm : TIME := T#100ms;
		sDSSOT2ProgNm : STRING[15] := 'DSSOT2';
		tDSSOT2RstDlyTm : TIME := T#0s;
		tDSSOT2SigInChkTm : TIME := T#100ms;
		sDSSOT3ProgNm : STRING[15] := 'DSSOT3';
		tDSSOT3RstDlyTm : TIME := T#0s;
		tDSSOT3SigInChkTm : TIME := T#100ms;
		bSOTReadyOnFirst : BOOL := TRUE;
		bShowMESName : BOOL := FALSE;
		bShowFMorMESActive : BOOL := FALSE;
		tyProdRcpMtrPshrExtSpd : tyUILmt := (diMax:=8,diMin:=1);
		tyProdRcpMtrPshrExtTorq : tyUILmt := (diMax:=100,diMin:=20);
		bProjUSFixToFixRail : BOOL := FALSE;
		bUIConvDirRL : BOOL := TRUE;
		bDSWidthChkPrep : BOOL := FALSE;
		bProjServoPullerPusherPrep : BOOL := FALSE;
		sPPProgNm : STRING[15] := 'ServoPullPusher';
		sPPDevice : STRING[3] := 'IF7';
		usiPPNode : USINT := 23;
		bPPDir : BOOL := FALSE;
		bPPDirBl : BOOL := FALSE;
		diPPPitchInUM : DINT := 3000;
		diPPMovBlDistInUM : DINT := 0;
		tyPPParamInHm : tyMotionCANParamInHm := (diStartVelInUMPS:=15000,diAcc:=25);
		tyPPParamInConvert : tyMotionCANParamInConvert := (diPitchInUM:=3000); (*estun1048576*)
		tyPPParam : tyMotionParam := (diAccInMS:=100,diDecInMS:=100,diAutoSpdInUMPS:=150000);
		tyPPTuning : tyMotionCANTuning := (diAsdaA2Inertia:=76,diAsdaA2PosLoopGain:=53,diAsdaA2PosFFGain:=50,diAsdaA2SpdLoopGain:=213,diAsdaA2SpdIntegral:=34,diAsdaA2LowPassFltr:=49,diAsdaA2AntiInterGain:=34,diAsdaA2FirstTorqueCmd:=300,diLex28LTNDderivativeGain_P800:=0,diLex28LTNIintegralGain_P801:=0,diLex28LTNIVdeIntlGain_P802:=0,diLex28LTNPpropotionalGain_P803:=0,diLex28LTNUSERGAIN_P804:=0,diLex28NLAFFLPFHZspringFil_P805:=0,diLex28NLFILTDAMPING_P814:=0,diLex28NLFILTT1_P815:=0,diPronetInertia:=0,diPronetRealTimeAutoAdjSet:=0,diPronetPosLoopGain:=0,diPronetSpdLoopGain:=0,diPronetSpdIntegral:=0,diPronetTorqueFilter:=0,diPronetPosFeedForward:=0,diPronetLowSpeedTestFiltering:=0,diPronetStopMode:=0);
		ePPServoMotorType : eServoMotorType := DeltaAsdaA2; (*Selection of  Motor Brand*)
		bProjFixClprMagDetectSenPrep : BOOL := FALSE;
		bCurtainSenPrep : BOOL := FALSE;
		bProjMagHeightChkPrep : BOOL := FALSE;
		diTravGoToMagWidthChkPt1 : DINT := 2000;
		diTravGoToMagWidthChkPt2 : DINT := 2000;
		diTravGoToMagWidthChkPt3 : DINT := 2000;
		bProjOutletShut2Prep : BOOL := FALSE;
		bProjOutletShut3Prep : BOOL := FALSE;
		bProjScanPrep : BOOL := FALSE;
		bProjOpConPrep : BOOL := FALSE;
		tyPPTorqParam : PPTorqParam := (usiStartTorque:=10,uiRatio:=478); (*Ratio= x/100*)
		bProjLifTravMnlLoad : BOOL := 0;
		eMidSenNcNoType : eMidSenParam := No;
		bHermesScannerPrep : BOOL := FALSE;
		bHermesSvyFirstMcInTheLine : BOOL := FALSE;
		bAutoRcpPrep : BOOL := FALSE;
		eCustomerReq : eCustomer := NA;
		bProjInletStopperPrep : BOOL := FALSE;
		sInletStopperProgNm : STRING[15] := 'Stopper A';
		bInletStopperTwoCtrlIn : BOOL := FALSE;
		tInletStopperExtDlyTm : TIME := T#1s;
		tInletStopperRetDlyTm : TIME := T#1s;
		eAutoRcpParamLmt : eAutoRcpLmt := (diMaxBottomCleranceInUM:=5500,diMaxTopClearamceInUM:=30000,diThicknessInUM:=6700);
		sAutoRcpProgNm : STRING[15] := 'AutoRcp';
		eAutoRcpPrecededBy : eAutoRcpPreceded := PrecededByF1;
		bChinesePrep : BOOL := FALSE;
		bGermanPrep : BOOL := FALSE;
		sHWInfoHMIMacAddress : STRING[27] := '00 - 60 - 65 - 82 - 0C - D7';
		tyUIBtnPosLmt : tyUILmt := (diMax:=1,diMin:=1);
	END_STRUCT;
	tyNtParamIn1 : 	STRUCT
		eAct : eNtParamAction;
		udiRstErr : UDINT;
		sFileName : STRING[80] := 'NutekParameter.dat';
		sProgNm : STRING[80] := 'NtParam';
		tyMpNtParamMpLink : MpComIdentType;
		sFileName1 : STRING[80] := 'NutekParameter.xml';
		sPVName : STRING[80] := 'NtParam:tyMpNtParamCurr1';
	END_STRUCT;
	tyNtParamOut1 : 	STRUCT
		eStat : eNtParamAction;
		eStatus : eFBStatus;
		sStatTxt : STRING[200];
		tyAlmData : tyAlmDat;
		bFileNotFound : BOOL;
	END_STRUCT;
	tyUILmt : 	STRUCT
		diMax : DINT;
		diMin : DINT;
	END_STRUCT;
	tyNtParamGen : 	STRUCT
		In : tyNtParamIn1;
		Out : tyNtParamOut1;
	END_STRUCT;
END_TYPE

(**)

TYPE
	PPTorqParam : 	STRUCT
		usiStartTorque : USINT;
		uiRatio : UINT;
	END_STRUCT;
END_TYPE

(*NtBosch China With Mid Sensor changed*)

TYPE
	eMidSenParam :
		(
		No,
		NcBoschChina
		);
	eCustomer :
		(
		NA,
		Bosch_China, (*Reject Mode notify When one Mag Full, Standard notify when two Mag full*)
		Bosch_Portugal,
		Bosch_America,
		Bosch_Malaysia,
		Siemens,
		We_Fabricate,
		New_Member5,
		New_Member6,
		New_Member7,
		New_Member8,
		New_Member9,
		New_Member10
		);
	eAutoRcpLmt : 	STRUCT
		diMaxBottomCleranceInUM : DINT;
		diMaxTopClearamceInUM : DINT;
		diThicknessInUM : DINT;
	END_STRUCT;
	eAutoRcpPreceded :
		(
		PrecededBySelf,
		PrecededByF1,
		PrecededByF2
		);
END_TYPE

(**)
```

### NtParam.var - Change By Project
```iecst
(**)
VAR
	g_tyNtParamCurr : tyNtParam;
	g_tyNtParamOut : tyNtParamOut1;
END_VAR
```

### Program Logical/NtParam/NtParam (IEC)

#### InputRef_Link.var
```iecst
(*2019-03-25*)
(**)
VAR
	p_bLinkStartupRun : REFERENCE TO BOOL;
	p_bSimu : REFERENCE TO BOOL;
END_VAR
```

#### Local.var
```iecst
(**)
VAR
	tylocalNtParam : tyNtParamGen;
	udiStatus : UDINT := 0;
	sStatTxt : STRING[200] := '';
	a_sStatText : ARRAY[0..50] OF STRING[200] := ['Idling','Creating Directory','Reading Files','Writing Files','Loading Data From XML','Saving Data To XML',45('')];
END_VAR
(**)
(*Local Alarm*)
VAR
	tyAlmData : tyAlmDat;
END_VAR
(*Local Output*)
VAR
	tyMpNtParamCurr1 : tyNtParam;
	bFileNotFound : BOOL;
END_VAR
(**)
(*Local Input*)
VAR
	udiRstErr : UDINT := 0;
	sFileName : STRING[80] := 'NutekParameter.dat';
	sProgNm : STRING[15] := 'NtParam';
	sFileName1 : STRING[80] := 'NutekParameter.xml';
	sPVName : STRING[100] := 'NtParam:tyMpNtParamCurr1';
	tyMpNtParamMpLink : MpComIdentType;
END_VAR
(**)
(*Local*)
VAR
	tyNtParamCurr : tyNtParam;
	bRstErr : BOOL;
	udiRstErrOld : UDINT;
	bInitDone : BOOL;
	bInitialDone : BOOL;
	usiStep : USINT;
	fbMpNtParamRegPar : MpRecipeRegPar;
	fbMpNtParamXml : MpRecipeXml;
	fbDirCreate1 : fbDirCreate;
	fbDirCreate2 : fbDirCreate;
	fbDirCreate3 : fbDirCreate;
	fbFileRead1 : fbFileFullReadEncry;
	fbFileWrite1 : fbFileFullWriteEncry;
	udiModuleNum : UDINT := 5151;
END_VAR
```

#### Act_Alarm.st
```iecst
ACTION Act_Alarm:

	IF tylocalNtParam.In.udiRstErr <> udiRstErrOld THEN
		bRstErr			:= TRUE;
		udiRstErrOld	:= tylocalNtParam.In.udiRstErr;
	ELSE
		bRstErr			:= FALSE;
	END_IF

	//Reset Error
	IF (tylocalNtParam.Out.eStatus = Error) AND bRstErr THEN
		tylocalNtParam.In.eAct	  := NtParamActIdle;
		tylocalNtParam.Out.eStat  := NtParamActIdle;
	END_IF

	//Reset Done
	IF tylocalNtParam.Out.eStatus = Done AND tylocalNtParam.In.eAct = NtParamActIdle THEN
		tylocalNtParam.Out.eStat 	:= NtParamActIdle;
	END_IF

	//Error
	IF EDGEPOS(tylocalNtParam.Out.eStatus = Error) THEN

		tylocalNtParam.Out.tyAlmData.udiCode		:= udiStatus;
		tylocalNtParam.Out.tyAlmData.eSeverity		:= AlmSeverityError;
		tylocalNtParam.Out.tyAlmData.udiRunTime	    := tylocalNtParam.Out.tyAlmData.udiRunTime + 1;
		tylocalNtParam.Out.tyAlmData.bAlm			:= TRUE;
		tylocalNtParam.Out.tyAlmData.udiModuleNum	:= udiModuleNum;
		g_tyAlmProgNm.sNtParamProgNm				:= sProgNm;

	ELSIF bRstErr AND (tylocalNtParam.Out.tyAlmData.udiCode <> 0) THEN

		tylocalNtParam.Out.tyAlmData.udiCode	:= 0;
		tylocalNtParam.Out.tyAlmData.eSeverity	:= AlmSeverityNA;
		tylocalNtParam.Out.tyAlmData.bAlm		:= FALSE;

		sStatTxt	:= a_sStatText[tylocalNtParam.Out.eStat];

	END_IF

END_ACTION
```

#### Act_InitGlobal.st
```iecst
(** 2019-03-25 **)
ACTION Act_InitGlobal:

	(* Always Change If Project Change *)

	//Pass Data To Link
	p_bLinkStartupRun ACCESS p_StartupRun;

	//Pass Data To Internal Use
	p_udiRstErr ACCESS p_RstErrReset;

	p_bSimu ACCESS p_UISimuMod;
	(* Always Change If Project Change *)

END_ACTION
```

#### Act_Initial.st
```iecst
ACTION Act_Initial:

	//Initial
	sStatTxt	:= a_sStatText[tylocalNtParam.Out.eStat];

	fbDirCreate1.sDevice	:= 'F';
	fbDirCreate1.sDirName	:= 'Private';
	fbDirCreate1(bEn := FALSE);

	fbDirCreate2.sDevice	:= 'Private';
	fbDirCreate2.sDirName	:= 'NutekParameter';
	fbDirCreate2(bEn := FALSE);

	fbDirCreate3.sDevice	:= 'Private';
	fbDirCreate3.sDirName	:= 'NutekParameterXml';
	fbDirCreate3(bEn := FALSE);

	fbFileRead1.sDevice			:= 'NtParam';
	fbFileRead1.sFile			:= tylocalNtParam.In.sFileName;
	fbFileRead1.udiOffset		:= 0;
	fbFileRead1.p_Dest			:= ADR(tyNtParamCurr);
	fbFileRead1.udiLen			:= SIZEOF(tyNtParamCurr);
	fbFileRead1.usiEncryptCode	:= 130;
	fbFileRead1(bEn := FALSE);

	fbFileWrite1.sDevice		:= 'NtParam';
	fbFileWrite1.sFile			:= tylocalNtParam.In.sFileName;
	fbFileWrite1.udiOffset		:= 0;
	fbFileWrite1.p_Src			:= ADR(tyNtParamCurr);
	fbFileWrite1.udiLen			:= SIZEOF(tyNtParamCurr);
	fbFileWrite1.udiOption		:= 0;
	fbFileWrite1.usiEncryptCode	:= 130;
	fbFileWrite1(bEn := FALSE);

	tyMpNtParamMpLink	:= gRecipeXml;

	fbMpNtParamRegPar.MpLink	:= ADR(tyMpNtParamMpLink);
	fbMpNtParamRegPar.PVName	:= ADR(tylocalNtParam.In.sPVName);
	fbMpNtParamRegPar(Enable := FALSE);

	fbMpNtParamXml.MpLink		:= ADR(tyMpNtParamMpLink);
	fbMpNtParamXml.DeviceName	:= ADR('MpNtParam');
	fbMpNtParamXml.FileName		:= ADR(tylocalNtParam.In.sFileName1);
	fbMpNtParamXml(Enable := FALSE);

END_ACTION
```

#### Act_InputConfig.st
```iecst
ACTION Act_InputConfig:

	tylocalNtParam.In.udiRstErr := g_tyRstErrOut.udiRstErr;

	IF g_tyStartUp.bRun THEN
		tylocalNtParam.In.eAct := g_tyStartUp.eNtParamAct;
	ELSE
		tylocalNtParam.In.eAct := tylocalNtParam.In.eAct;
	END_IF

END_ACTION
```

#### Act_LinkAction.st
```iecst
(** 2019-04-09 **)
ACTION Act_LinkAction:

	IF p_bLinkStartupRun = TRUE THEN
		p_eAct ACCESS p_StartupNtParamAct;
	ELSIF p_bSimu THEN
		p_eAct ACCESS p_UINtWr;
	ELSE
		p_eAct ACCESS ADR(eAct);
	END_IF

END_ACTION
```

#### Act_Main.st
```iecst
ACTION Act_Main:

	IF tylocalNtParam.Out.eStatus = Idle THEN
		tylocalNtParam.Out.eStat	:= tylocalNtParam.In.eAct;
	END_IF

	//Main
	CASE tylocalNtParam.Out.eStat OF

		NtParamActIdle:
			IF tylocalNtParam.Out.eStatus <> Idle THEN	//Reset Data
				//Private
				fbDirCreate1(bEn := FALSE);
				fbDirCreate2(bEn := FALSE);
				fbDirCreate3(bEn := FALSE);
				fbFileRead1(bEn := FALSE);
				fbFileWrite1(bEn := FALSE);
				fbMpNtParamRegPar(Enable := FALSE);
				fbMpNtParamXml(Enable := FALSE);
				usiStep	:= 0;

				tylocalNtParam.Out.bFileNotFound	:= FALSE;

				sStatTxt	:= a_sStatText[tylocalNtParam.Out.eStat];

			END_IF

			tylocalNtParam.Out.eStatus	:= Idle;

		NtParamActCreateDir:
			IF tylocalNtParam.Out.eStatus = Idle OR tylocalNtParam.Out.eStatus = Busy THEN

				tylocalNtParam.Out.eStatus	:= Busy;

				sStatTxt	:= a_sStatText[tylocalNtParam.Out.eStat];

				CASE usiStep OF
					0:
						fbDirCreate1(bEn := TRUE);
						IF fbDirCreate1.udiStatus = 0 THEN
							usiStep	:= 1;
						ELSIF fbDirCreate1.udiStatus < 65534 THEN
							tylocalNtParam.Out.eStatus		:= Error;

							IF fbDirCreate1.udiStatus = 1908 THEN
								udiStatus	:= 10000;	//Create User Directory Error
							ELSE
								udiStatus	:= fbDirCreate1.udiStatus;
							END_IF
						END_IF

					1:
						fbDirCreate2(bEn := TRUE);
						IF fbDirCreate2.udiStatus = 0 THEN
							usiStep	:= 2;
						ELSIF fbDirCreate2.udiStatus < 65534 THEN
							tylocalNtParam.Out.eStatus		:= Error;

							IF fbDirCreate2.udiStatus = 1908 THEN
								udiStatus	:= 10001;	//Create Nutek Parameter Directory Error
							ELSE
								udiStatus	:= fbDirCreate2.udiStatus;
							END_IF
						END_IF

					2:
						fbDirCreate3(bEn := TRUE);
						IF fbDirCreate3.udiStatus = 0 THEN
							tylocalNtParam.Out.eStatus	:= Done;
						ELSIF fbDirCreate3.udiStatus < 65534 THEN
							tylocalNtParam.Out.eStatus		:= Error;

							IF fbDirCreate3.udiStatus = 1908 THEN
								udiStatus	:= 10014;	//Create Nutek Parameter xml Directory Error
							ELSE
								udiStatus	:= fbDirCreate3.udiStatus;
							END_IF
						END_IF

				END_CASE

			END_IF

		NtParamActWrite:
			IF tylocalNtParam.Out.eStatus = Idle OR tylocalNtParam.Out.eStatus = Busy THEN

				tylocalNtParam.Out.eStatus	:= Busy;

				sStatTxt	:= a_sStatText[tylocalNtParam.Out.eStat];

				fbFileWrite1(bEn := TRUE);
				IF fbFileWrite1.udiStatus = 0 THEN
					tylocalNtParam.Out.eStatus	:= Done;
				ELSIF fbFileWrite1.udiStatus < 65534 THEN
					tylocalNtParam.Out.eStatus	:= Error;

					IF fbFileWrite1.udiStatus = 1900 THEN
						udiStatus	:= 10002;	//File Open Error While Writing
					ELSIF fbFileWrite1.udiStatus = 1901 THEN
						udiStatus	:= 10003;	//File Create Error While Writing
					ELSIF fbFileWrite1.udiStatus = 1903 THEN
						udiStatus	:= 10004;	//File Write Error
					ELSIF fbFileWrite1.udiStatus = 1904 THEN
						udiStatus	:= 10005;	//File Close Error While Writing
					ELSIF fbFileWrite1.udiStatus = 1914 THEN
						udiStatus	:= 10009;	//Directory Does Not Exist While Writing
					ELSE
						udiStatus	:= fbFileWrite1.udiStatus;
					END_IF
				END_IF

			END_IF

		NtParamActRead:
			IF tylocalNtParam.Out.eStatus = Idle OR tylocalNtParam.Out.eStatus = Busy THEN

				tylocalNtParam.Out.eStatus	:= Busy;

				sStatTxt	:= a_sStatText[tylocalNtParam.Out.eStat];

				fbFileRead1(bEn := TRUE);
				IF fbFileRead1.udiStatus = 0 THEN
					tylocalNtParam.Out.eStatus	:= Done;
				ELSIF fbFileRead1.udiStatus < 65534 THEN
					tylocalNtParam.Out.eStatus := Error;

					IF fbFileRead1.udiStatus = 1900 THEN
						udiStatus	:= 10006;	//File Open Error While Reading
					ELSIF fbFileRead1.udiStatus = 1902 THEN
						udiStatus	:= 10007;	//File Read Error
					ELSIF fbFileRead1.udiStatus = 1904 THEN
						udiStatus	:= 10008;	//File Close Error While Reading
					ELSIF fbFileRead1.udiStatus = 1915 THEN
						tylocalNtParam.Out.eStatus			:= Done;
						tylocalNtParam.Out.bFileNotFound	:= TRUE;
					ELSE
						udiStatus	:= fbFileRead1.udiStatus;
					END_IF
				END_IF

			END_IF

		NtParamActLoad:
			IF tylocalNtParam.Out.eStatus = Idle OR tylocalNtParam.Out.eStatus = Busy THEN

				tylocalNtParam.Out.eStatus	:= Busy;

				sStatTxt	:= a_sStatText[tylocalNtParam.Out.eStat];

				CASE usiStep OF
					0:
						fbMpNtParamRegPar(Enable := TRUE);

						IF (fbMpNtParamRegPar.Active = TRUE) AND (fbMpNtParamRegPar.StatusID = 0) THEN
							usiStep	:= 1;
						ELSIF fbMpNtParamRegPar.StatusID <> 0 THEN
							tylocalNtParam.Out.eStatus		:= Error;
							udiStatus						:= 10010;	//MpRecipeRegPar Error While Loading
						END_IF

					1:
						fbMpNtParamXml.Load	:= TRUE;
						fbMpNtParamXml.Save	:= FALSE;
						fbMpNtParamXml(Enable := TRUE);

						IF (fbMpNtParamXml.Active = TRUE) AND (fbMpNtParamXml.CommandDone = TRUE) AND (fbMpNtParamXml.StatusID = 0) THEN
							//	tylocalNtParam.Out.eStatus	:= Done;
							usiStep	:= 2;
							tyNtParamCurr	:= tyMpNtParamCurr1;
						ELSIF fbMpNtParamXml.StatusID <> 0 THEN
							tylocalNtParam.Out.eStatus		:= Error;
							udiStatus						:= 10011;	//MpRecipeXml Error While Loading
						END_IF

					2:
						fbFileWrite1(bEn := TRUE);
						IF fbFileWrite1.udiStatus = 0 THEN
							tylocalNtParam.Out.eStatus	 := Done;
						ELSIF fbFileWrite1.udiStatus < 65534 THEN
							tylocalNtParam.Out.eStatus	 := Error;

							IF fbFileWrite1.udiStatus = 1900 THEN
								udiStatus	:= 10002;	//File Open Error While Writing
							ELSIF fbFileWrite1.udiStatus = 1901 THEN
								udiStatus	:= 10003;	//File Create Error While Writing
							ELSIF fbFileWrite1.udiStatus = 1903 THEN
								udiStatus	:= 10004;	//File Write Error
							ELSIF fbFileWrite1.udiStatus = 1904 THEN
								udiStatus	:= 10005;	//File Close Error While Writing
							ELSIF fbFileWrite1.udiStatus = 1914 THEN
								udiStatus	:= 10009;	//Directory Does Not Exist While Writing
							ELSE
								udiStatus	:= fbFileWrite1.udiStatus;
							END_IF
						END_IF

				END_CASE

			END_IF

		NtParamActSave:
			IF tylocalNtParam.Out.eStatus = Idle OR tylocalNtParam.Out.eStatus = Busy THEN

				tylocalNtParam.Out.eStatus	:= Busy;

				sStatTxt	:= a_sStatText[tylocalNtParam.Out.eStat];

				CASE usiStep OF
					0:
						tyMpNtParamCurr1	:= tyNtParamCurr;
						fbMpNtParamRegPar(Enable := TRUE);

						IF (fbMpNtParamRegPar.Active = TRUE) AND (fbMpNtParamRegPar.StatusID = 0) THEN
							usiStep	:= 1;
						ELSIF fbMpNtParamRegPar.StatusID <> 0 THEN
							tylocalNtParam.Out.eStatus		:= Error;
							udiStatus	:= 10012;	//MpRecipeRegPar Error While Saving
						END_IF

					1:
						fbMpNtParamXml.Load	:= FALSE;
						fbMpNtParamXml.Save	:= TRUE;
						fbMpNtParamXml(Enable := TRUE);

						IF (fbMpNtParamXml.Active = TRUE) AND (fbMpNtParamXml.CommandDone = TRUE) AND (fbMpNtParamXml.StatusID = 0) THEN
							tylocalNtParam.Out.eStatus	:= Done;
						ELSIF fbMpNtParamXml.StatusID <> 0 THEN
							tylocalNtParam.Out.eStatus		:= Error;
							udiStatus	:= 10013;	//MpRecipeXml Error While Saving
						END_IF

				END_CASE

			END_IF

	END_CASE

END_ACTION
```

#### Act_OutputConfig.st
```iecst
ACTION Act_OutputConfig:

	g_tyNtParamCurr := tyNtParamCurr;
	g_tyNtParamOut  := tylocalNtParam.Out;

END_ACTION
```

#### Cyclic.st
```iecst
PROGRAM _CYCLIC

	IF bInitialDone = FALSE THEN
		bInitialDone	:= TRUE;
		Act_Initial;

	ELSE
		Act_InputConfig;
		Act_Main;
		Act_OutputConfig;
		Act_Alarm;

	END_IF

END_PROGRAM
```

#### Init.st
```iecst
(** 2019-05-20 **)
PROGRAM _INIT

	(* Always Change If Project Change *)

	//Pass Address To Global Address For External Use
	//Action, State & Status
	p_NtParamStat						:= ADR(eStat);
	p_NtParamStatus						:= ADR(eStatus);
	p_NtParamStatTxt					:= ADR(sStatTxt);

	//Alarm
	p_NtParamAlmData					:= ADR(tyAlmData);

	//Output
	p_NtParamFileNotFound				:= ADR(bFileNotFound);

	p_NtParamCurr						:= ADR(tyNtParamCurr);

	p_NtParamDISettings					:= ADR(tyNtParamCurr.tyDISettings);
	p_NtParamDOSettings					:= ADR(tyNtParamCurr.tyDOSettings);
	p_NtParamAWPushPulPrep				:= ADR(tyNtParamCurr.bAWPusherPrep);
	p_NtParamAWPrep						:= ADR(tyNtParamCurr.bAWPrep);
	p_NtParamLFPrep						:= ADR(tyNtParamCurr.bLFPrep);
	p_NtParamLeaderMc					:= ADR(tyNtParamCurr.bLeaderMc);
	p_NtParamLFUsrSetPrep				:= ADR(tyNtParamCurr.bLFUsrSetPrep);
	p_NtParamLFWidth2Prep				:= ADR(tyNtParamCurr.bLFProdWidth2Prep);
	p_NtParamLFWidthLimit				:= ADR(tyNtParamCurr.diLFWidthLimit);
	p_NtParamLFProdWidthChk				:= ADR(tyNtParamCurr.bLFProdWidthChk);
	p_NtParamUSWidthChkPrep				:= ADR(tyNtParamCurr.bUSWidthChkPrep);
	p_NtParamLCSLFPrep					:= ADR(tyNtParamCurr.bLCSLFPrep);
	p_NtParamLCSReqRcpPrep				:= ADR(tyNtParamCurr.bLCSReqRcpPrep);
	p_NtParamLCSManageRcpPrep			:= ADR(tyNtParamCurr.bLCSManageRcpPrep);
	p_NtParamLCSLiveDatPrep				:= ADR(tyNtParamCurr.bLCSLiveDatPrep);
	p_NtParamIPCSMEMA9851ExtdPrep		:= ADR(tyNtParamCurr.bIPCSMEMA9851ExtdPrep);
	p_NtParamVSMEMAPrep					:= ADR(tyNtParamCurr.bVSMEMAPrep);
	p_NtParamHermesPrep					:= ADR(tyNtParamCurr.bHermesPrep);
	p_NtParamHermesRmtPrep				:= ADR(tyNtParamCurr.bHermesRmtPrep);
	p_NtParamOvenInfoPrep				:= ADR(tyNtParamCurr.bOvenInfoPrep);
	p_NtParamOvenInfoExtdPrep			:= ADR(tyNtParamCurr.bOvenInfoExtdPrep);
	p_NtParamSSaverPrep					:= ADR(tyNtParamCurr.bSSaverPrep);
	p_NtParamWidthOffset				:= ADR(tyNtParamCurr.diWidthOffsetInUM);
	p_NtParamPushPulAWidthOffset		:= ADR(tyNtParamCurr.diAWPushPulOffsetInUM);
	p_NtParamJobNo						:= ADR(tyNtParamCurr.sJobNo);
	p_NtParamNtAddr						:= ADR(tyNtParamCurr.usiNtAddr);
	p_NtParamShutterWaitTmr				:= ADR(tyNtParamCurr.tShutterWaitTmr);
	p_NtParamProjAIVInPosSenPrep		:= ADR(tyNtParamCurr.bProjAIVInPosSenPrep);
	p_NtParamProjMagBuffferActLoad		:= ADR(tyNtParamCurr.eProjMagBuffferActLoad);
	p_NtParamProjLifterMagPlatform		:= ADR(tyNtParamCurr.bProjLifterMagPlatform);

	p_NtParamProjLaneBPrep				:= ADR(tyNtParamCurr.bProjLaneBPrep);
	p_NtParamProjBrdPerSltPrep			:= ADR(tyNtParamCurr.bProjBrdPerSltPrep);
	p_NtParamProjLongBrdPrep			:= ADR(tyNtParamCurr.bProjLongBrdPrep);
	p_NtParamProjInletShutPrep			:= ADR(tyNtParamCurr.bProjInletShutPrep);
	p_NtParamProjOutletShutPrep			:= ADR(tyNtParamCurr.bProjOutletShutPrep);
	p_NtParamProjOutletShut2Prep		:= ADR(tyNtParamCurr.bProjOutletShut2Prep);
	p_NtParamProjOutletShut3Prep		:= ADR(tyNtParamCurr.bProjOutletShut3Prep);
	p_NtParamProjStopperAPrep			:= ADR(tyNtParamCurr.bProjStopperAPrep);
	p_NtParamProjStopperBPrep			:= ADR(tyNtParamCurr.bProjStopperBPrep);
	p_NtParamProjMag1ConvPrep			:= ADR(tyNtParamCurr.bProjMag1ConvPrep);
	p_NtParamProjMag2ConvPrep			:= ADR(tyNtParamCurr.bProjMag2ConvPrep);
	p_NtParamProjMag3ConvPrep			:= ADR(tyNtParamCurr.bProjMag3ConvPrep);
	p_NtParamProjMagOrientChkSenPrep	:= ADR(tyNtParamCurr.bProjMagOrientChkSenPrep);
	p_NtParamProjAGVPrep				:= ADR(tyNtParamCurr.bProjAGVPrep);
	p_NtParamProjTCPAGVSigPrep			:= ADR(tyNtParamCurr.bProjTCPAGVSigPrep);
	p_NtParamProjBypsInitConvPrep		:= ADR(tyNtParamCurr.bProjBypsInitConvPrep);
	p_NtParamProjRlsNewProdPrep			:= ADR(tyNtParamCurr.bProjRlsNewProdPrep);
	p_NtParamProjBtnInsertRmvMag		:= ADR(tyNtParamCurr.bProjBtnInsertRmvMag);
	p_NtParamProjMagMinSlt				:= ADR(tyNtParamCurr.diProjMagMinSlt);
	p_NtParamProjMagMaxSlt				:= ADR(tyNtParamCurr.diProjMagMaxSlt);
	p_NtParamProjMag					:= ADR(tyNtParamCurr.eProjMag);
	p_NtParamProjConvDir				:= ADR(tyNtParamCurr.eProjConvDir);
	p_NtParamProjMagConvDir				:= ADR(tyNtParamCurr.eProjMagConvDir);
	p_NtParamProjMagAutoVerifyPrep		:= ADR(tyNtParamCurr.bMagAutoVerifyPrep);
	p_NtParamProjMotorizedPusherPrep	:= ADR(tyNtParamCurr.bProjMotorizedPusherPrep);
	p_NtParamProjMagAWPrep				:= ADR(tyNtParamCurr.bProjMagAWPrep);
	p_NtParamProjMagSafetyBarPrep		:= ADR(tyNtParamCurr.bProjMagSafetyBarPrep);
	p_NtParamProjFixClpMagDSenPrep		:= ADR(tyNtParamCurr.bProjFixClprMagDetectSenPrep);

	p_NtParamProjLifter2Prep			:= ADR(tyNtParamCurr.bProjLifter2Prep);
	p_NtParamProjMagConvLane1Prep		:= ADR(tyNtParamCurr.bProjMagConvLane1Prep); //MagConv Lane1 ,2
	p_NtParamProjMagConvLane2Prep		:= ADR(tyNtParamCurr.bProjMagConvLane2Prep);
	p_NtParamProjInMagConvDir			:= ADR(tyNtParamCurr.eProjInMagConvDir);
	p_NtParamProjOutMagConvDir			:= ADR(tyNtParamCurr.eProjOutMagConvDir);
	p_NtParamProjLifterMagConvDir		:= ADR(tyNtParamCurr.eProjLifterMagConvDir);
	p_NtParamProjInMagConv2Dir			:= ADR(tyNtParamCurr.eProjInMagConv2Dir);
	p_NtParamProjOutMagConv2Dir			:= ADR(tyNtParamCurr.eProjOutMagConv2Dir);
	p_NtParamProjLifterMagConv2Dir		:= ADR(tyNtParamCurr.eProjLifterMagConv2Dir);

	p_NtParamProjTopEntStprPrep			:= ADR(tyNtParamCurr.bProjTopEntStprPrep);
	p_NtParamProjTopMidStprPrep			:= ADR(tyNtParamCurr.bProjTopMidStprPrep);
	p_NtParamProjTopExtStprPrep			:= ADR(tyNtParamCurr.bProjTopExtStprPrep);
	p_NtParamProjBtmMidStprPrep			:= ADR(tyNtParamCurr.bProjBtmMidStprPrep);
	p_NtParamProjBtmExtStprPrep			:= ADR(tyNtParamCurr.bProjBtmExtStprPrep);
	p_NtParamProjTopEntStprPrep2			:= ADR(tyNtParamCurr.bProjTopEntStprPrep2);
	p_NtParamProjTopMidStprPrep2			:= ADR(tyNtParamCurr.bProjTopMidStprPrep2);
	p_NtParamProjTopExtStprPrep2			:= ADR(tyNtParamCurr.bProjTopExtStprPrep2);
	p_NtParamProjBtmMidStprPrep2			:= ADR(tyNtParamCurr.bProjBtmMidStprPrep2);
	p_NtParamProjBtmExtStprPrep2			:= ADR(tyNtParamCurr.bProjBtmExtStprPrep2);

	p_NtParamTopEntStprProgNm			:= ADR(tyNtParamCurr.sTopEntStprProgNm); //Lane1 top zone stopper
	p_NtParamTopEntStprTwoCtrlIn		:= ADR(tyNtParamCurr.bTopEntStprTwoCtrlIn);
	p_NtParamTopEntStprExtDlyTm			:= ADR(tyNtParamCurr.tTopEntStprExtDlyTm);
	p_NtParamTopEntStprRetDlyTm			:= ADR(tyNtParamCurr.tTopEntStprRetDlyTm);
	p_NtParamTopMidStprProgNm			:= ADR(tyNtParamCurr.sTopMidStprProgNm);
	p_NtParamTopMidStprTwoCtrlIn		:= ADR(tyNtParamCurr.bTopMidStprTwoCtrlIn);
	p_NtParamTopMidStprExtDlyTm			:= ADR(tyNtParamCurr.tTopMidStprExtDlyTm);
	p_NtParamTopMidStprRetDlyTm			:= ADR(tyNtParamCurr.tTopMidStprRetDlyTm);
	p_NtParamTopExtStprProgNm			:= ADR(tyNtParamCurr.sTopExtStprProgNm);
	p_NtParamTopExtStprTwoCtrlIn		:= ADR(tyNtParamCurr.bTopExtStprTwoCtrlIn);
	p_NtParamTopExtStprExtDlyTm			:= ADR(tyNtParamCurr.tTopExtStprExtDlyTm);
	p_NtParamTopExtStprRetDlyTm			:= ADR(tyNtParamCurr.tTopExtStprRetDlyTm);
	p_NtParamBtmMidStprProgNm			:= ADR(tyNtParamCurr.sBtmMidStprProgNm);
	p_NtParamBtmMidStprTwoCtrlIn		:= ADR(tyNtParamCurr.bBtmMidStprTwoCtrlIn);
	p_NtParamBtmMidStprExtDlyTm			:= ADR(tyNtParamCurr.tBtmMidStprExtDlyTm);
	p_NtParamBtmMidStprRetDlyTm			:= ADR(tyNtParamCurr.tBtmMidStprRetDlyTm);
	p_NtParamBtmExtStprProgNm			:= ADR(tyNtParamCurr.sBtmExtStprProgNm);
	p_NtParamBtmExtStprTwoCtrlIn		:= ADR(tyNtParamCurr.bBtmExtStprTwoCtrlIn);
	p_NtParamBtmExtStprExtDlyTm			:= ADR(tyNtParamCurr.tBtmExtStprExtDlyTm);
	p_NtParamBtmExtStprRetDlyTm			:= ADR(tyNtParamCurr.tBtmExtStprRetDlyTm);

	p_NtParamTopEntStprProgNm2				:= ADR(tyNtParamCurr.sTopEntStprProgNm2); //Lane2 top zone stopper
	p_NtParamTopEntStprTwoCtrlIn2			:= ADR(tyNtParamCurr.bTopEntStprTwoCtrlIn2);
	p_NtParamTopEntStprExtDlyTm2			:= ADR(tyNtParamCurr.tTopEntStprExtDlyTm2);
	p_NtParamTopEntStprRetDlyTm2			:= ADR(tyNtParamCurr.tTopEntStprRetDlyTm2);
	p_NtParamTopMidStprProgNm2				:= ADR(tyNtParamCurr.sTopMidStprProgNm2);
	p_NtParamTopMidStprTwoCtrlIn2			:= ADR(tyNtParamCurr.bTopMidStprTwoCtrlIn2);
	p_NtParamTopMidStprExtDlyTm2			:= ADR(tyNtParamCurr.tTopMidStprExtDlyTm2);
	p_NtParamTopMidStprRetDlyTm2			:= ADR(tyNtParamCurr.tTopMidStprRetDlyTm2);
	p_NtParamTopExtStprProgNm2				:= ADR(tyNtParamCurr.sTopExtStprProgNm2);
	p_NtParamTopExtStprTwoCtrlIn2			:= ADR(tyNtParamCurr.bTopExtStprTwoCtrlIn2);
	p_NtParamTopExtStprExtDlyTm2			:= ADR(tyNtParamCurr.tTopExtStprExtDlyTm2);
	p_NtParamTopExtStprRetDlyTm2			:= ADR(tyNtParamCurr.tTopExtStprRetDlyTm2);
	p_NtParamBtmMidStprProgNm2				:= ADR(tyNtParamCurr.sBtmMidStprProgNm2);
	p_NtParamBtmMidStprTwoCtrlIn2			:= ADR(tyNtParamCurr.bBtmMidStprTwoCtrlIn2);
	p_NtParamBtmMidStprExtDlyTm2			:= ADR(tyNtParamCurr.tBtmMidStprExtDlyTm2);
	p_NtParamBtmMidStprRetDlyTm2			:= ADR(tyNtParamCurr.tBtmMidStprRetDlyTm2);
	p_NtParamBtmExtStprProgNm2				:= ADR(tyNtParamCurr.sBtmExtStprProgNm2);
	p_NtParamBtmExtStprTwoCtrlIn2			:= ADR(tyNtParamCurr.bBtmExtStprTwoCtrlIn2);
	p_NtParamBtmExtStprExtDlyTm2			:= ADR(tyNtParamCurr.tBtmExtStprExtDlyTm2);
	p_NtParamBtmExtStprRetDlyTm2			:= ADR(tyNtParamCurr.tBtmExtStprRetDlyTm2);

	p_NtParamInMagConvProgNm			:= ADR(tyNtParamCurr.sInMagConvProgNm); //InMag, OutMag, LifterMag Lane1
	p_NtParamInMagConvOnDirMod			:= ADR(tyNtParamCurr.bInMagConvOnDirMod);
	p_NtParamInMagConvMtrOffDlyTm		:= ADR(tyNtParamCurr.tInMagConvMtrOffDlyTm);
	p_NtParamOutMagConvProgNm			:= ADR(tyNtParamCurr.sOutMagConvProgNm);
	p_NtParamOutMagConvOnDirMod			:= ADR(tyNtParamCurr.bOutMagConvOnDirMod);
	p_NtParamOutMagConvMtrOffDlyTm		:= ADR(tyNtParamCurr.tOutMagConvMtrOffDlyTm);
	p_NtParamLifterMagProgNm			:= ADR(tyNtParamCurr.sLifterMagProgNm);
	p_NtParamLifterMagOnDirMod			:= ADR(tyNtParamCurr.bLifterMagOnDirMod);
	p_NtParamLifterMagMtrOffDlyTm		:= ADR(tyNtParamCurr.tLifterMagMtrOffDlyTm);
	p_NtParamLifterMagClprClampTO		:= ADR(tyNtParamCurr.tLifterMagClprClampTO);
	p_NtParamLifterMagClprUnclampTO		:= ADR(tyNtParamCurr.tLifterMagClprUnclampTO);
	p_NtParamInMagConv2ProgNm			:= ADR(tyNtParamCurr.sInMagConv2ProgNm); //InMag, OutMag, LifterMag Lane2
	p_NtParamInMagConv2OnDirMod			:= ADR(tyNtParamCurr.bInMagConv2OnDirMod);
	p_NtParamInMagConv2MtrOffDlyTm		:= ADR(tyNtParamCurr.tInMagConv2MtrOffDlyTm);
	p_NtParamOutMagConv2ProgNm			:= ADR(tyNtParamCurr.sOutMagConv2ProgNm);
	p_NtParamOutMagConv2OnDirMod		:= ADR(tyNtParamCurr.bOutMagConv2OnDirMod);
	p_NtParamOutMagConv2MtrOffDlyTm		:= ADR(tyNtParamCurr.tOutMagConv2MtrOffDlyTm);
	p_NtParamLifterMag2ProgNm			:= ADR(tyNtParamCurr.sLifterMag2ProgNm);
	p_NtParamLifterMag2OnDirMod			:= ADR(tyNtParamCurr.bLifterMag2OnDirMod);
	p_NtParamLifterMag2MtrOffDlyTm		:= ADR(tyNtParamCurr.tLifterMag2MtrOffDlyTm);
	p_NtParamLifterMagClprClampTO2		:= ADR(tyNtParamCurr.tLifterMagClprClampTO2);
	p_NtParamLifterMagClprUnclampTO2		:= ADR(tyNtParamCurr.tLifterMagClprUnclampTO2); //##

	p_NtParamUsrFolderProgNm			:= ADR(tyNtParamCurr.sUsrFolderProgNm);
	p_NtParamLibVersionProgNm			:= ADR(tyNtParamCurr.sLibVersionProgNm);
	p_NtParamTimeProgNm					:= ADR(tyNtParamCurr.sTimeProgNm);

	p_NtParamHWInfoProgNm				:= ADR(tyNtParamCurr.sHWInfoProgNm);
	p_NtParamHWInfoDevice				:= ADR(tyNtParamCurr.sHWInfoDevice);

	p_NtParamTLBuzMode					:= ADR(tyNtParamCurr.eTLBuzMode);

	p_NtParamTLChgRcpBlinkTm		:= ADR(tyNtParamCurr.tTLChgRcpBlinkTm);

	p_NtParamTLErrBlinkTm			:= ADR(tyNtParamCurr.tTLErrBlinkTm);
	p_NtParamBuzErrOnTm				:= ADR(tyNtParamCurr.tBuzErrOnTm);
	p_NtParamBuzErrRestTm			:= ADR(tyNtParamCurr.tBuzErrRestTm);
	p_NtParamBuzErrOnCntr			:= ADR(tyNtParamCurr.usiBuzErrOnCntr);
	p_NtParamBuzErrStopSeqEn		:= ADR(tyNtParamCurr.bBuzErrStopSeqEn);
	p_NtParamBuzErrStopSeqCntr		:= ADR(tyNtParamCurr.usiBuzErrStopSeqCntr);

	p_NtParamTLWarnBlinkTm			:= ADR(tyNtParamCurr.tTLWarnBlinkTm);
	p_NtParamBuzWarnOnTm			:= ADR(tyNtParamCurr.tBuzWarnOnTm);
	p_NtParamBuzWarnRestTm			:= ADR(tyNtParamCurr.tBuzWarnRestTm);
	p_NtParamBuzWarnOnCntr			:= ADR(tyNtParamCurr.usiBuzWarnOnCntr);
	p_NtParamBuzWarnStopSeqEn		:= ADR(tyNtParamCurr.bBuzWarnStopSeqEn);
	p_NtParamBuzWarnStopSeqCntr		:= ADR(tyNtParamCurr.usiBuzWarnStopSeqCntr);

	p_NtParamTLWarn1BlinkTm			:= ADR(tyNtParamCurr.tTLWarn1BlinkTm);
	p_NtParamBuzWarn1OnTm			:= ADR(tyNtParamCurr.tBuzWarn1OnTm);
	p_NtParamBuzWarn1RestTm			:= ADR(tyNtParamCurr.tBuzWarn1RestTm);
	p_NtParamBuzWarn1OnCntr			:= ADR(tyNtParamCurr.usiBuzWarn1OnCntr);
	p_NtParamBuzWarn1StopSeqEn		:= ADR(tyNtParamCurr.bBuzWarn1StopSeqEn);
	p_NtParamBuzWarn1StopSeqCntr	:= ADR(tyNtParamCurr.usiBuzWarn1StopSeqCntr);

	p_NtParamTLWarn2BlinkTm			:= ADR(tyNtParamCurr.tTLWarn2BlinkTm);
	p_NtParamBuzWarn2OnTm			:= ADR(tyNtParamCurr.tBuzWarn2OnTm);
	p_NtParamBuzWarn2RestTm			:= ADR(tyNtParamCurr.tBuzWarn2RestTm);
	p_NtParamBuzWarn2OnCntr			:= ADR(tyNtParamCurr.usiBuzWarn2OnCntr);
	p_NtParamBuzWarn2StopSeqEn		:= ADR(tyNtParamCurr.bBuzWarn2StopSeqEn);
	p_NtParamBuzWarn2StopSeqCntr	:= ADR(tyNtParamCurr.usiBuzWarn2StopSeqCntr);

	p_NtParamTLWarn3BlinkTm			:= ADR(tyNtParamCurr.tTLWarn3BlinkTm);
	p_NtParamBuzWarn3OnTm			:= ADR(tyNtParamCurr.tBuzWarn3OnTm);
	p_NtParamBuzWarn3RestTm			:= ADR(tyNtParamCurr.tBuzWarn3RestTm);
	p_NtParamBuzWarn3OnCntr			:= ADR(tyNtParamCurr.usiBuzWarn3OnCntr);
	p_NtParamBuzWarn3StopSeqEn		:= ADR(tyNtParamCurr.bBuzWarn3StopSeqEn);
	p_NtParamBuzWarn3StopSeqCntr	:= ADR(tyNtParamCurr.usiBuzWarn3StopSeqCntr);

	p_NtParamTLWarn4BlinkTm			:= ADR(tyNtParamCurr.tTLWarn4BlinkTm);
	p_NtParamBuzWarn4OnTm			:= ADR(tyNtParamCurr.tBuzWarn4OnTm);
	p_NtParamBuzWarn4RestTm			:= ADR(tyNtParamCurr.tBuzWarn4RestTm);
	p_NtParamBuzWarn4OnCntr			:= ADR(tyNtParamCurr.usiBuzWarn4OnCntr);
	p_NtParamBuzWarn4StopSeqEn		:= ADR(tyNtParamCurr.bBuzWarn4StopSeqEn);
	p_NtParamBuzWarn4StopSeqCntr	:= ADR(tyNtParamCurr.usiBuzWarn4StopSeqCntr);

	p_NtParamTLWarn5BlinkTm			:= ADR(tyNtParamCurr.tTLWarn5BlinkTm);
	p_NtParamBuzWarn5OnTm			:= ADR(tyNtParamCurr.tBuzWarn5OnTm);
	p_NtParamBuzWarn5RestTm			:= ADR(tyNtParamCurr.tBuzWarn5RestTm);
	p_NtParamBuzWarn5OnCntr			:= ADR(tyNtParamCurr.usiBuzWarn5OnCntr);
	p_NtParamBuzWarn5StopSeqEn		:= ADR(tyNtParamCurr.bBuzWarn5StopSeqEn);
	p_NtParamBuzWarn5StopSeqCntr	:= ADR(tyNtParamCurr.usiBuzWarn5StopSeqCntr);

	p_NtParamBuzAlertOnTm			:= ADR(tyNtParamCurr.tBuzAlertOnTm);
	p_NtParamBuzAlertRestTm			:= ADR(tyNtParamCurr.tBuzAlertRestTm);
	p_NtParamBuzAlertOnCntr			:= ADR(tyNtParamCurr.usiBuzAlertOnCntr);
	p_NtParamBuzAlertStopSeqEn		:= ADR(tyNtParamCurr.bBuzAlertStopSeqEn);
	p_NtParamBuzAlertStopSeqCntr	:= ADR(tyNtParamCurr.usiBuzAlertStopSeqCntr);

	p_NtParamTLBlueBlinkTm			:= ADR(tyNtParamCurr.tTLBlueBlinkTm);
	p_NtParamTLAmberBlinkTm			:= ADR(tyNtParamCurr.tTLAmberBlinkTm);
	p_NtParamTLWhiteBlinkTm			:= ADR(tyNtParamCurr.tTLWhiteBlinkTm);
	p_NtParamTLRedBlinkTm			:= ADR(tyNtParamCurr.tTLRedBlinkTm);
	p_NtParamTLGreenBlinkTm			:= ADR(tyNtParamCurr.tTLGreenBlinkTm);

	p_NtParamAlmProgNm					:= ADR(tyNtParamCurr.sAlmProgNm);
	p_NtParamAlmFileKeepDay				:= ADR(tyNtParamCurr.udiAlmFileKeepDay);

	p_NtParamProdRcpProgNm				:= ADR(tyNtParamCurr.sProdRcpProgNm);
	p_NtParamProdRcpListFileNm			:= ADR(tyNtParamCurr.sProdRcpListFileNm);
	p_NtParamProdRcpSingleFileNm		:= ADR(tyNtParamCurr.sProdRcpSingleFileNm);

	p_NtParamMpProdRcpProgNm			:= ADR(tyNtParamCurr.sMpProdRcpProgNm);
	p_NtParamMpProdRcpFileNm			:= ADR(tyNtParamCurr.sMpProdRcpFileNm);
	p_NtParamMpProdRcpPVNm				:= ADR(tyNtParamCurr.sMpProdRcpPVNm);

	p_NtParamMagRcpProgNm				:= ADR(tyNtParamCurr.sMagRcpProgNm);
	p_NtParamMagRcpListFileNm			:= ADR(tyNtParamCurr.sMagRcpListFileNm);
	p_NtParamMagRcpSingleFileNm			:= ADR(tyNtParamCurr.sMagRcpSingleFileNm);

	p_NtParamMcParamProgNm				:= ADR(tyNtParamCurr.sMcParamProgNm);
	p_NtParamMcParamFileNm				:= ADR(tyNtParamCurr.sMcParamFileNm);

	p_NtParamUsrMgmtProgNm				:= ADR(tyNtParamCurr.sUsrMgmtProgNm);

	p_NtParamBffr1ProgNm				:= ADR(tyNtParamCurr.sBffr1ProgNm);
	p_NtParamBffr1FileNm				:= ADR(tyNtParamCurr.sBffr1FileNm);
	p_NtParamBffr1NxtLoadSeq			:= ADR(tyNtParamCurr.bBffr1NxtLoadSeq);

	p_NtParamBffr2ProgNm				:= ADR(tyNtParamCurr.sBffr2ProgNm);
	p_NtParamBffr2FileNm				:= ADR(tyNtParamCurr.sBffr2FileNm);
	p_NtParamBffr2NxtLoadSeq			:= ADR(tyNtParamCurr.bBffr2NxtLoadSeq);

	p_NtParamBffr3ProgNm				:= ADR(tyNtParamCurr.sBffr3ProgNm);
	p_NtParamBffr3FileNm				:= ADR(tyNtParamCurr.sBffr3FileNm);
	p_NtParamBffr3NxtLoadSeq			:= ADR(tyNtParamCurr.bBffr3NxtLoadSeq);

	p_NtParamUSSMEMAAProgNm				:= ADR(tyNtParamCurr.sUSSMEMAAProgNm);
	p_NtParamUSSMEMAARstDlyTm			:= ADR(tyNtParamCurr.tUSSMEMAARstDlyTm);
	p_NtParamUSSMEMAASigInChkTm			:= ADR(tyNtParamCurr.tUSSMEMAASigInChkTm);

	p_NtParamUSSMEMABProgNm				:= ADR(tyNtParamCurr.sUSSMEMABProgNm);
	p_NtParamUSSMEMABRstDlyTm			:= ADR(tyNtParamCurr.tUSSMEMABRstDlyTm);
	p_NtParamUSSMEMABSigInChkTm			:= ADR(tyNtParamCurr.tUSSMEMABSigInChkTm);

	p_NtParamUSSMEMA1ProgNm				:= ADR(tyNtParamCurr.sUSSMEMA1ProgNm);
	p_NtParamUSSMEMA1RstDlyTm			:= ADR(tyNtParamCurr.tUSSMEMA1RstDlyTm);
	p_NtParamUSSMEMA1SigInChkTm			:= ADR(tyNtParamCurr.tUSSMEMA1SigInChkTm);

	p_NtParamUSSMEMA2ProgNm				:= ADR(tyNtParamCurr.sUSSMEMA2ProgNm);
	p_NtParamUSSMEMA2RstDlyTm			:= ADR(tyNtParamCurr.tUSSMEMA2RstDlyTm);
	p_NtParamUSSMEMA2SigInChkTm			:= ADR(tyNtParamCurr.tUSSMEMA2SigInChkTm);

	p_NtParamUSSMEMA3ProgNm				:= ADR(tyNtParamCurr.sUSSMEMA3ProgNm);
	p_NtParamUSSMEMA3RstDlyTm			:= ADR(tyNtParamCurr.tUSSMEMA3RstDlyTm);
	p_NtParamUSSMEMA3SigInChkTm			:= ADR(tyNtParamCurr.tUSSMEMA3SigInChkTm);

	p_NtParamDSSMEMA1ProgNm				:= ADR(tyNtParamCurr.sDSSMEMA1ProgNm);
	p_NtParamDSSMEMA1RstDlyTm			:= ADR(tyNtParamCurr.tDSSMEMA1RstDlyTm);
	p_NtParamDSSMEMA1SigInChkTm			:= ADR(tyNtParamCurr.tDSSMEMA1SigInChkTm);

	p_NtParamDSSMEMA2ProgNm				:= ADR(tyNtParamCurr.sDSSMEMA2ProgNm);
	p_NtParamDSSMEMA2RstDlyTm			:= ADR(tyNtParamCurr.tDSSMEMA2RstDlyTm);
	p_NtParamDSSMEMA2SigInChkTm			:= ADR(tyNtParamCurr.tDSSMEMA2SigInChkTm);

	p_NtParamDSSMEMA3ProgNm				:= ADR(tyNtParamCurr.sDSSMEMA3ProgNm);
	p_NtParamDSSMEMA3RstDlyTm			:= ADR(tyNtParamCurr.tDSSMEMA3RstDlyTm);
	p_NtParamDSSMEMA3SigInChkTm			:= ADR(tyNtParamCurr.tDSSMEMA3SigInChkTm);

	p_NtParamInShutterProgNm			:= ADR(tyNtParamCurr.sInShutterProgNm);
	p_NtParamInShutterTwoCtrlIn			:= ADR(tyNtParamCurr.bInShutterTwoCtrlIn);
	p_NtParamInShutterExtTO				:= ADR(tyNtParamCurr.tInShutterExtTO);
	p_NtParamInShutterRetTO				:= ADR(tyNtParamCurr.tInShutterRetTO);

	p_NtParamOutShutterProgNm			:= ADR(tyNtParamCurr.sOutShutterProgNm);
	p_NtParamOutShutterTwoCtrlIn		:= ADR(tyNtParamCurr.bOutShutterTwoCtrlIn);
	p_NtParamOutShutterExtTO			:= ADR(tyNtParamCurr.tOutShutterExtTO);
	p_NtParamOutShutterRetTO			:= ADR(tyNtParamCurr.tOutShutterRetTO);

	p_NtParamInletStopperProgNm				:= ADR(tyNtParamCurr.sInletStopperProgNm);
	p_NtParamInletStopperTwoCtrlIn			:= ADR(tyNtParamCurr.bInletStopperTwoCtrlIn);
	p_NtParamInletStopperExtDlyTm			:= ADR(tyNtParamCurr.tInletStopperExtDlyTm);
	p_NtParamInletStopperRetDlyTm			:= ADR(tyNtParamCurr.tInletStopperRetDlyTm);

	p_NtParamStopperAProgNm				:= ADR(tyNtParamCurr.sStopperAProgNm);
	p_NtParamStopperATwoCtrlIn			:= ADR(tyNtParamCurr.bStopperATwoCtrlIn);
	p_NtParamStopperAExtDlyTm			:= ADR(tyNtParamCurr.tStopperAExtDlyTm);
	p_NtParamStopperARetDlyTm			:= ADR(tyNtParamCurr.tStopperARetDlyTm);

	p_NtParamStopperBProgNm				:= ADR(tyNtParamCurr.sStopperBProgNm);
	p_NtParamStopperBTwoCtrlIn			:= ADR(tyNtParamCurr.bStopperBTwoCtrlIn);
	p_NtParamStopperBExtDlyTm			:= ADR(tyNtParamCurr.tStopperBExtDlyTm);
	p_NtParamStopperBRetDlyTm			:= ADR(tyNtParamCurr.tStopperBRetDlyTm);

	p_NtParamPshrConvProgNm				:= ADR(tyNtParamCurr.sPshrConvProgNm);
	p_NtParamPshrConvOnDirMod			:= ADR(tyNtParamCurr.bPshrConvOnDirMod);
	p_NtParamPshrConvMtrOffDlyTm		:= ADR(tyNtParamCurr.tPshrConvMtrOffDlyTm);
	p_NtParamPshrConvPshrExtTO			:= ADR(tyNtParamCurr.tPshrConvPshrExtTO);
	p_NtParamPshrConvPshrRetTO			:= ADR(tyNtParamCurr.tPshrConvPshrRetTO);

	p_NtParamMagConv1ProgNm				:= ADR(tyNtParamCurr.sMagConv1ProgNm);
	p_NtParamMagConv1OnDirMod			:= ADR(tyNtParamCurr.bMagConv1OnDirMod);
	p_NtParamMagConv1MtrOffDlyTm		:= ADR(tyNtParamCurr.tMagConv1MtrOffDlyTm);
	p_NtParamMagConv1ClprClampTO		:= ADR(tyNtParamCurr.tMagConv1ClprClampTO);
	p_NtParamMagConv1ClprUnclampTO		:= ADR(tyNtParamCurr.tMagConv1ClprUnclampTO);

	p_NtParamMagConv2ProgNm				:= ADR(tyNtParamCurr.sMagConv2ProgNm);
	p_NtParamMagConv2OnDirMod			:= ADR(tyNtParamCurr.bMagConv2OnDirMod);
	p_NtParamMagConv2MtrOffDlyTm		:= ADR(tyNtParamCurr.tMagConv2MtrOffDlyTm);
	p_NtParamMagConv2ClprClampTO		:= ADR(tyNtParamCurr.tMagConv2ClprClampTO);
	p_NtParamMagConv2ClprUnclampTO		:= ADR(tyNtParamCurr.tMagConv2ClprUnclampTO);

	p_NtParamMagConv3ProgNm				:= ADR(tyNtParamCurr.sMagConv3ProgNm);
	p_NtParamMagConv3OnDirMod			:= ADR(tyNtParamCurr.bMagConv3OnDirMod);
	p_NtParamMagConv3MtrOffDlyTm		:= ADR(tyNtParamCurr.tMagConv3MtrOffDlyTm);
	p_NtParamMagConv3ClprClampTO		:= ADR(tyNtParamCurr.tMagConv3ClprClampTO);
	p_NtParamMagConv3ClprUnclampTO		:= ADR(tyNtParamCurr.tMagConv3ClprUnclampTO);

	p_NtParamMag1SafetyBarProgNm		:= ADR(tyNtParamCurr.sMag1SafetyBarProgNm);
	p_NtParamMag1SafetyBarTwoCtrlIn		:= ADR(tyNtParamCurr.bMag1SafetyBarTwoCtrlIn);
	p_NtParamMag1SafetyBarExtTO			:= ADR(tyNtParamCurr.tMag1SafetyBarExtTO);
	p_NtParamMag1SafetyBarRetTO			:= ADR(tyNtParamCurr.tMag1SafetyBarRetTO);

	p_NtParamMag2SafetyBarProgNm		:= ADR(tyNtParamCurr.sMag2SafetyBarProgNm);
	p_NtParamMag2SafetyBarTwoCtrlIn		:= ADR(tyNtParamCurr.bMag2SafetyBarTwoCtrlIn);
	p_NtParamMag2SafetyBarExtTO			:= ADR(tyNtParamCurr.tMag2SafetyBarExtTO);
	p_NtParamMag2SafetyBarRetTO			:= ADR(tyNtParamCurr.tMag2SafetyBarRetTO);

	p_NtParamMag3SafetyBarProgNm		:= ADR(tyNtParamCurr.sMag3SafetyBarProgNm);
	p_NtParamMag3SafetyBarTwoCtrlIn		:= ADR(tyNtParamCurr.bMag3SafetyBarTwoCtrlIn);
	p_NtParamMag3SafetyBarExtTO			:= ADR(tyNtParamCurr.tMag3SafetyBarExtTO);
	p_NtParamMag3SafetyBarRetTO			:= ADR(tyNtParamCurr.tMag3SafetyBarRetTO);

	p_NtParamMag1AWEngageProgNm			:= ADR(tyNtParamCurr.sMag1AWEngageProgNm);
	p_NtParamMag1AWEngageTwoCtrlIn		:= ADR(tyNtParamCurr.bMag1AWEngageTwoCtrlIn);
	p_NtParamMag1AWEngageExtTO			:= ADR(tyNtParamCurr.tMag1AWEngageExtTO);
	p_NtParamMag1AWEngageRetTO			:= ADR(tyNtParamCurr.tMag1AWEngageRetTO);

	p_NtParamMag2AWEngageProgNm			:= ADR(tyNtParamCurr.sMag2AWEngageProgNm);
	p_NtParamMag2AWEngageTwoCtrlIn		:= ADR(tyNtParamCurr.bMag2AWEngageTwoCtrlIn);
	p_NtParamMag2AWEngageExtTO			:= ADR(tyNtParamCurr.tMag2AWEngageExtTO);
	p_NtParamMag2AWEngageRetTO			:= ADR(tyNtParamCurr.tMag2AWEngageRetTO);

	p_NtParamMag3AWEngageProgNm			:= ADR(tyNtParamCurr.sMag3AWEngageProgNm);
	p_NtParamMag3AWEngageTwoCtrlIn		:= ADR(tyNtParamCurr.bMag3AWEngageTwoCtrlIn);
	p_NtParamMag3AWEngageExtTO			:= ADR(tyNtParamCurr.tMag3AWEngageExtTO);
	p_NtParamMag3AWEngageRetTO			:= ADR(tyNtParamCurr.tMag3AWEngageRetTO);

	p_NtParamMtrPshrProgNm				:= ADR(tyNtParamCurr.sMtrPshrProgNm);
	p_NtParamMtrPshrDir					:= ADR(tyNtParamCurr.bMtrPshrDir);
	p_NtParamMtrPshrAlmRstTm			:= ADR(tyNtParamCurr.tMtrPshrAlmRstTm);
	p_NtParamMtrPshrAlmTrigTm			:= ADR(tyNtParamCurr.tMtrPshrAlmTrigTm);
	p_NtParamMtrPshrExtTO				:= ADR(tyNtParamCurr.tMtrPshrExtTO);
	p_NtParamMtrPshrRetTO				:= ADR(tyNtParamCurr.tMtrPshrRetTO);
	p_NtParamMtrPshrExtSlowSpd			:= ADR(tyNtParamCurr.diMtrPshrExtSlowSpd);
	p_NtParamMtrPshrRetSlowSpd			:= ADR(tyNtParamCurr.diMtrPshrRetSlowSpd);
	p_NtParamMtrPshrExtNomSpd			:= ADR(tyNtParamCurr.diMtrPshrExtNomSpd);
	p_NtParamMtrPshrRetNomSpd			:= ADR(tyNtParamCurr.diMtrPshrRetNomSpd);
	p_NtParamMtrPshrExtTorq				:= ADR(tyNtParamCurr.diMtrPshrRetNomSpd);
	p_NtParamMtrPshrRetTorq				:= ADR(tyNtParamCurr.diMtrPshrRetTorq);
	p_NtParamMtrPshrStartTorq			:= ADR(tyNtParamCurr.diMtrPshrStartTorq);

	p_NtParamAWPushPulProgNm			:= ADR(tyNtParamCurr.sAWPushPullProgNm);
	p_NtParamAWPushPulDevice			:= ADR(tyNtParamCurr.sAWPushPullDevice);
	p_NtParamAWPushPulNode				:= ADR(tyNtParamCurr.usiAWPushPullNode);
	p_NtParamAWPushPulDir				:= ADR(tyNtParamCurr.bAWPushPullDir);
	p_NtParamAWPushPulDirBl				:= ADR(tyNtParamCurr.bAWPushPullDirBl);
	p_NtParamAWPushPulPitchInUM			:= ADR(tyNtParamCurr.diAWPushPullPitchInUM);
	p_NtParamAWPushPulMovBlDistInUM		:= ADR(tyNtParamCurr.diAWPushPullMovBlDistInUM);
	p_NtParamAWPushPulParamInHm			:= ADR(tyNtParamCurr.tyAWPushPullParamInHm);
	p_NtParamAWPushPulParamInConvert	:= ADR(tyNtParamCurr.tyAWPushPullParamInConvert);
	p_NtParamAWPushPulParam				:= ADR(tyNtParamCurr.tyAWPushPullParam);
	p_NtParamAWPushPulAcc				:= ADR(tyNtParamCurr.tyAWPushPullParam.diAccInMS);
	p_NtParamAWPushPulDec				:= ADR(tyNtParamCurr.tyAWPushPullParam.diDecInMS);
	p_NtParamAWPushPulAutoSpd			:= ADR(tyNtParamCurr.tyAWPushPullParam.diAutoSpdInUMPS);
	p_NtParamAWPushPulTuning			:= ADR(tyNtParamCurr.tyAWPushPullTuning);
	p_NtParamAWPushPulMotorType			:= ADR(tyNtParamCurr.eAWPushPullServoMotorType);

	p_NtParamAWProgNm					:= ADR(tyNtParamCurr.sAWProgNm);
	p_NtParamAWDevice					:= ADR(tyNtParamCurr.sAWDevice);
	p_NtParamAWNode						:= ADR(tyNtParamCurr.usiAWNode);
	p_NtParamAWDir						:= ADR(tyNtParamCurr.bAWDir);
	p_NtParamAWDirBl					:= ADR(tyNtParamCurr.bAWDirBl);
	p_NtParamAWPitchInUM				:= ADR(tyNtParamCurr.diAWPitchInUM);
	p_NtParamAWMovBlDistInUM			:= ADR(tyNtParamCurr.diAWMovBlDistInUM);
	p_NtParamAWParamInHm				:= ADR(tyNtParamCurr.tyAWParamInHm);
	p_NtParamAWParamInConvert			:= ADR(tyNtParamCurr.tyAWParamInConvert);
	p_NtParamAWParam					:= ADR(tyNtParamCurr.tyAWParam);
	p_NtParamAWAcc						:= ADR(tyNtParamCurr.tyAWParam.diAccInMS);
	p_NtParamAWDec						:= ADR(tyNtParamCurr.tyAWParam.diDecInMS);
	p_NtParamAWAutoSpd					:= ADR(tyNtParamCurr.tyAWParam.diAutoSpdInUMPS);
	p_NtParamAWTuning					:= ADR(tyNtParamCurr.tyAWTuning);
	p_NtParamAWMotorType				:= ADR(tyNtParamCurr.eAWServoMotorType);

	p_NtParamTravProgNm					:= ADR(tyNtParamCurr.sTravProgNm);
	p_NtParamTravDevice					:= ADR(tyNtParamCurr.sTravDevice);
	p_NtParamTravNode					:= ADR(tyNtParamCurr.usiTravNode);
	p_NtParamTravDir					:= ADR(tyNtParamCurr.bTravDir);
	p_NtParamTravParamInHm				:= ADR(tyNtParamCurr.tyTravParamInHm);
	p_NtParamTravParamInConvert			:= ADR(tyNtParamCurr.tyTravParamInConvert);
	p_NtParamTravParam					:= ADR(tyNtParamCurr.tyTravParam);
	p_NtParamTravAcc					:= ADR(tyNtParamCurr.tyTravParam.diAccInMS);
	p_NtParamTravDec					:= ADR(tyNtParamCurr.tyTravParam.diDecInMS);
	p_NtParamTravAutoSpd				:= ADR(tyNtParamCurr.tyTravParam.diAutoSpdInUMPS);
	p_NtParamTravLongBrdAutoSpd			:= ADR(tyNtParamCurr.diTravAutoSpdLongBrdInUMPS);
	p_NtParamTravMotorType				:= ADR(tyNtParamCurr.eTravServoMotorType);
	p_NtParamTravTuning					:= ADR(tyNtParamCurr.tyTravTuning);

	p_NtParamLifterProgNm				:= ADR(tyNtParamCurr.sLifterProgNm);
	p_NtParamLifterDevice				:= ADR(tyNtParamCurr.sLifterDevice);
	p_NtParamLifterNode					:= ADR(tyNtParamCurr.usiLifterNode);
	p_NtParamLifterDir					:= ADR(tyNtParamCurr.bLifterDir);
	p_NtParamLifterParamInHm			:= ADR(tyNtParamCurr.tyLifterParamInHm);
	p_NtParamLifterParamInConvert		:= ADR(tyNtParamCurr.tyLifterParamInConvert);
	p_NtParamLifterParam				:= ADR(tyNtParamCurr.tyLifterParam);
	p_NtParamLifterAcc					:= ADR(tyNtParamCurr.tyLifterParam.diAccInMS);
	p_NtParamLifterDec					:= ADR(tyNtParamCurr.tyLifterParam.diDecInMS);
	p_NtParamLifterAutoSpd				:= ADR(tyNtParamCurr.tyLifterParam.diAutoSpdInUMPS);
	p_NtParamLifterTuning				:= ADR(tyNtParamCurr.tyLifterTuning);
	p_NtParamLifterMotorType			:= ADR(tyNtParamCurr.eLifterServoMotorType);

	p_NtParamLifter2ProgNm				:= ADR(tyNtParamCurr.sLifterProgNm2);
	p_NtParamLifter2Device				:= ADR(tyNtParamCurr.sLifterDevice2);
	p_NtParamLifter2Node				:= ADR(tyNtParamCurr.usiLifterNode2);
	p_NtParamLifter2Dir					:= ADR(tyNtParamCurr.bLifterDir2);
	p_NtParamLifter2ParamInHm			:= ADR(tyNtParamCurr.tyLifterParamInHm2);
	p_NtParamLifter2ParamInConvert		:= ADR(tyNtParamCurr.tyLifterParamInConvert2);
	p_NtParamLifter2Param				:= ADR(tyNtParamCurr.tyLifterParam2);
	p_NtParamLifter2Acc					:= ADR(tyNtParamCurr.tyLifterParam2.diAccInMS);
	p_NtParamLifter2Dec					:= ADR(tyNtParamCurr.tyLifterParam2.diDecInMS);
	p_NtParamLifter2AutoSpd				:= ADR(tyNtParamCurr.tyLifterParam2.diAutoSpdInUMPS);
	p_NtParamLifter2Tuning				:= ADR(tyNtParamCurr.tyLifterTuning2);
	p_NtParamLifter2MotorType			:= ADR(tyNtParamCurr.eLifterServoMotorType2);

	p_NtParamDIProgNm					:= ADR(tyNtParamCurr.sDIProgNm);

	p_NtParamAGVProgNm					:= ADR(tyNtParamCurr.sAGVProgNm);

	p_NtParamAGVMag1ProgNm				:= ADR(tyNtParamCurr.sAGVMag1ProgNm);

	p_NtParamAGVMag2ProgNm				:= ADR(tyNtParamCurr.sAGVMag2ProgNm);

	p_NtParamAGVMag3ProgNm				:= ADR(tyNtParamCurr.sAGVMag3ProgNm);

	p_NtParamHermesProgNm				:= ADR(tyNtParamCurr.sHermesProgNm);
	p_NtParamHermesRetainFileNm			:= ADR(tyNtParamCurr.sHermesRetainFileNm);
	p_NtParamHermesConfigFileNm			:= ADR(tyNtParamCurr.sHermesConfigFileNm);

	p_NtParamUSHermesAProgNm			:= ADR(tyNtParamCurr.sUSHermesAProgNm);
	p_NtParamUSHermesAFileKeepDay		:= ADR(tyNtParamCurr.udiUSHermesAFileKeepDay);
	p_NtParamUSHermesAAliveTmInSec		:= ADR(tyNtParamCurr.udiUSHermesAAliveTmInSec);
	p_NtParamUSHermesAConnTO			:= ADR(tyNtParamCurr.tUSHermesAConnTO);

	p_NtParamUSHermesBProgNm			:= ADR(tyNtParamCurr.sUSHermesBProgNm);
	p_NtParamUSHermesBFileKeepDay		:= ADR(tyNtParamCurr.udiUSHermesBFileKeepDay);
	p_NtParamUSHermesBAliveTmInSec		:= ADR(tyNtParamCurr.udiUSHermesBAliveTmInSec);
	p_NtParamUSHermesBConnTO			:= ADR(tyNtParamCurr.tUSHermesBConnTO);

	p_NtParamRmtHermesProgNm			:= ADR(tyNtParamCurr.sRmtHermesProgNm);
	p_NtParamRmtHermesConfigFileNm		:= ADR(tyNtParamCurr.sRmtHermesConfigFileNm);
	p_NtParamRmtHermesFileKeepDay		:= ADR(tyNtParamCurr.udiRmtHermesFileKeepDay);
	p_NtParamRmtHermesAliveTmInSec		:= ADR(tyNtParamCurr.udiRmtHermesAliveTmInSec);
	p_NtParamRmtHermesSndBffrSize		:= ADR(tyNtParamCurr.udiRmtHermesSndBffrSize);
	p_NtParamRmtHermesRcvBffrSize		:= ADR(tyNtParamCurr.udiRmtHermesRcvBffrSize);

	p_NtParamLFLeaderProgNm				:= ADR(tyNtParamCurr.sLFLeaderProgNm);
	p_NtParamLFLeaderOnlineChkDlyTm		:= ADR(tyNtParamCurr.tLFLeaderOnlineChkDlyTm);
	p_NtParamLFLeaderSetTmOffDlyTm		:= ADR(tyNtParamCurr.tLFLeaderSetTmOffDlyTm);

	p_NtParamLFFllowerOnlineChkDlyTm:= ADR(tyNtParamCurr.tLFFollowerOnlineChkDlyTm);
	p_NtParamLFFollowerProgNm			:= ADR(tyNtParamCurr.sLFFollowerProgNm);

	p_NtParamFollower1ProgNm			:= ADR(tyNtParamCurr.sFollower1ProgNm);
	p_NtParamFollower2ProgNm			:= ADR(tyNtParamCurr.sFollower2ProgNm);

	p_NtParamLCSProgNm					:= ADR(tyNtParamCurr.sLCSProgNm);

	p_NtParamLCSMngRcpProgNm			:= ADR(tyNtParamCurr.sLCSMngRcpProgNm);

	p_NtParamLCSLFProgNm				:= ADR(tyNtParamCurr.sLCSLFProgNm);

	p_NtParamOpsTravLifULProgNm			:= ADR(tyNtParamCurr.sOpsTravLifULProgNm);

	p_NtParamOpsMagUL1ProgNm			:= ADR(tyNtParamCurr.sOpsMagUL1ProgNm);

	p_NtParamOpsMagUL2ProgNm			:= ADR(tyNtParamCurr.sOpsMagUL2ProgNm);

	p_NtParamOpsMagUL3ProgNm			:= ADR(tyNtParamCurr.sOpsMagUL3ProgNm);

	p_NtParamOpsMagConvUL1ProgNm		:= ADR(tyNtParamCurr.sOpsMagConvUL1ProgNm);

	p_NtParamOpsMagConvUL2ProgNm		:= ADR(tyNtParamCurr.sOpsMagConvUL2ProgNm);

	p_NtParamOpsMagConvUL3ProgNm		:= ADR(tyNtParamCurr.sOpsMagConvUL3ProgNm);

	p_NtParamOpsMagConvStprProgNm		:= ADR(tyNtParamCurr.sOpsMagConvStprProgNm);
	p_NtParamOpsMagConvStprProgNm1		:= ADR(tyNtParamCurr.sOpsMagConvStprProgNm1);

	p_NtParamProdRcpMinWidth			:= ADR(tyNtParamCurr.tyProdRcpWidth.diMin);
	p_NtParamProdRcpMaxWidth			:= ADR(tyNtParamCurr.tyProdRcpWidth.diMax);
	p_NtParamProdRcpMinMinSlt			:= ADR(tyNtParamCurr.tyProdRcpMinSlt.diMin);
	p_NtParamProdRcpMaxMinSlt			:= ADR(tyNtParamCurr.tyProdRcpMinSlt.diMax);
	p_NtParamProdRcpMinMaxSlt			:= ADR(tyNtParamCurr.tyProdRcpMaxSlt.diMin);
	p_NtParamProdRcpMaxMaxSlt			:= ADR(tyNtParamCurr.tyProdRcpMaxSlt.diMax);
	p_NtParamProdRcpMinPitch			:= ADR(tyNtParamCurr.tyProdRcpPitch.diMin);
	p_NtParamProdRcpMaxPitch			:= ADR(tyNtParamCurr.tyProdRcpPitch.diMax);
	p_NtParamProdRcpMinBrdPerSlt		:= ADR(tyNtParamCurr.tyProdRcpBrdPerSlt.diMin);
	p_NtParamProdRcpMaxBrdPerSlt		:= ADR(tyNtParamCurr.tyProdRcpBrdPerSlt.diMax);
	p_NtParamProdRcpMinMcModA			:= ADR(tyNtParamCurr.tyProdRcpMcModA.diMin);
	p_NtParamProdRcpMaxMcModA			:= ADR(tyNtParamCurr.tyProdRcpMcModA.diMax);
	p_NtParamProdRcpMinMcModAB			:= ADR(tyNtParamCurr.tyProdRcpMcModAB.diMin);
	p_NtParamProdRcpMaxMcModAB			:= ADR(tyNtParamCurr.tyProdRcpMcModAB.diMax);
	p_NtParamProdRcpMinMinReqFrBffr		:= ADR(tyNtParamCurr.tyProdRcpOvenMinReqFreeBffr.diMin);
	p_NtParamProdRcpMaxMinReqFrBffr		:= ADR(tyNtParamCurr.tyProdRcpOvenMinReqFreeBffr.diMax);

	p_NtParamSelClamp1ProgNm			:= ADR(tyNtParamCurr.sSelClamp1ProgNm);
	p_NtParamSelClamp1TwoCtrlIn			:= ADR(tyNtParamCurr.bSelClamp1TwoCtrlIn);
	p_NtParamSelClamp1ExtDlyTm			:= ADR(tyNtParamCurr.tSelClamp1ExtDlyTm);
	p_NtParamSelClamp1RetDlyTm			:= ADR(tyNtParamCurr.tSelClamp1RetDlyTm);

	p_NtParamSelClamp2ProgNm			:= ADR(tyNtParamCurr.sSelClamp2ProgNm);
	p_NtParamSelClamp2TwoCtrlIn			:= ADR(tyNtParamCurr.bSelClamp2TwoCtrlIn);
	p_NtParamSelClamp2ExtDlyTm			:= ADR(tyNtParamCurr.tSelClamp2ExtDlyTm);
	p_NtParamSelClamp2RetDlyTm			:= ADR(tyNtParamCurr.tSelClamp2RetDlyTm);

	p_NtParamSelClamp3ProgNm			:= ADR(tyNtParamCurr.sSelClamp3ProgNm);
	p_NtParamSelClamp3TwoCtrlIn			:= ADR(tyNtParamCurr.bSelClamp3TwoCtrlIn);
	p_NtParamSelClamp3ExtDlyTm			:= ADR(tyNtParamCurr.tSelClamp3ExtDlyTm);
	p_NtParamSelClamp3RetDlyTm			:= ADR(tyNtParamCurr.tSelClamp3RetDlyTm);

	p_NtParamMagAW1ProgNm				:= ADR(tyNtParamCurr.sMagAW1ProgNm);
	p_NtParamMagAW1Device				:= ADR(tyNtParamCurr.sMagAW1Device);
	p_NtParamMagAW1Node					:= ADR(tyNtParamCurr.usiMagAW1Node);
	p_NtParamMagAW1Dir					:= ADR(tyNtParamCurr.bMagAW1Dir);
	p_NtParamMagAW1DirBl				:= ADR(tyNtParamCurr.bMagAW1DirBl);
	p_NtParamMagAW1PitchInUM			:= ADR(tyNtParamCurr.diMagAW1PitchInUM);
	p_NtParamMagAW1MovBlDistInUM		:= ADR(tyNtParamCurr.diMagAW1MovBlDistInUM);
	p_NtParamMagAW1ParamInHm			:= ADR(tyNtParamCurr.tyMagAW1ParamInHm);
	p_NtParamMagAW1ParamInConvert		:= ADR(tyNtParamCurr.tyMagAW1ParamInConvert);
	p_NtParamMagAW1Param				:= ADR(tyNtParamCurr.tyMagAW1Param);
	p_NtParamMagAW1Acc					:= ADR(tyNtParamCurr.tyMagAW1Param.diAccInMS);
	p_NtParamMagAW1Dec					:= ADR(tyNtParamCurr.tyMagAW1Param.diDecInMS);
	p_NtParamMagAW1AutoSpd				:= ADR(tyNtParamCurr.tyMagAW1Param.diAutoSpdInUMPS);
	p_NtParamMagAW1Tuning				:= ADR(tyNtParamCurr.tyMagAW1Tuning);
	p_NtParamMagAW1EngageSpdInUMPS		:= ADR(tyNtParamCurr.diMagAW1EngageSpdInUMPS);
	p_NtParamMagAW1MotorType			:= ADR(tyNtParamCurr.eMagAW1ServoMotorType);
	p_NtParamMag1WidthOffset			:= ADR(tyNtParamCurr.diMag1WidthOffsetInUM);

	p_NtParamMagAW2ProgNm				:= ADR(tyNtParamCurr.sMagAW2ProgNm);
	p_NtParamMagAW2Device				:= ADR(tyNtParamCurr.sMagAW2Device);
	p_NtParamMagAW2Node					:= ADR(tyNtParamCurr.usiMagAW2Node);
	p_NtParamMagAW2Dir					:= ADR(tyNtParamCurr.bMagAW2Dir);
	p_NtParamMagAW2DirBl				:= ADR(tyNtParamCurr.bMagAW2DirBl);
	p_NtParamMagAW2PitchInUM			:= ADR(tyNtParamCurr.diMagAW2PitchInUM);
	p_NtParamMagAW2MovBlDistInUM		:= ADR(tyNtParamCurr.diMagAW2MovBlDistInUM);
	p_NtParamMagAW2ParamInHm			:= ADR(tyNtParamCurr.tyMagAW2ParamInHm);
	p_NtParamMagAW2ParamInConvert		:= ADR(tyNtParamCurr.tyMagAW2ParamInConvert);
	p_NtParamMagAW2Param				:= ADR(tyNtParamCurr.tyMagAW2Param);
	p_NtParamMagAW2Acc					:= ADR(tyNtParamCurr.tyMagAW2Param.diAccInMS);
	p_NtParamMagAW2Dec					:= ADR(tyNtParamCurr.tyMagAW2Param.diDecInMS);
	p_NtParamMagAW2AutoSpd				:= ADR(tyNtParamCurr.tyMagAW2Param.diAutoSpdInUMPS);
	p_NtParamMagAW2Tuning				:= ADR(tyNtParamCurr.tyMagAW2Tuning);
	p_NtParamMagAW2EngageSpdInUMPS		:= ADR(tyNtParamCurr.diMagAW2EngageSpdInUMPS);
	p_NtParamMagAW2MotorType			:= ADR(tyNtParamCurr.eMagAW2ServoMotorType);
	p_NtParamMag2WidthOffset			:= ADR(tyNtParamCurr.diMag2WidthOffsetInUM);

	p_NtParamMagAW3ProgNm				:= ADR(tyNtParamCurr.sMagAW3ProgNm);
	p_NtParamMagAW3Device				:= ADR(tyNtParamCurr.sMagAW3Device);
	p_NtParamMagAW3Node					:= ADR(tyNtParamCurr.usiMagAW3Node);
	p_NtParamMagAW3Dir					:= ADR(tyNtParamCurr.bMagAW3Dir);
	p_NtParamMagAW3DirBl				:= ADR(tyNtParamCurr.bMagAW3DirBl);
	p_NtParamMagAW3PitchInUM			:= ADR(tyNtParamCurr.diMagAW3PitchInUM);
	p_NtParamMagAW3MovBlDistInUM		:= ADR(tyNtParamCurr.diMagAW3MovBlDistInUM);
	p_NtParamMagAW3ParamInHm			:= ADR(tyNtParamCurr.tyMagAW3ParamInHm);
	p_NtParamMagAW3ParamInConvert		:= ADR(tyNtParamCurr.tyMagAW3ParamInConvert);
	p_NtParamMagAW3Param				:= ADR(tyNtParamCurr.tyMagAW3Param);
	p_NtParamMagAW3Acc					:= ADR(tyNtParamCurr.tyMagAW3Param.diAccInMS);
	p_NtParamMagAW3Dec					:= ADR(tyNtParamCurr.tyMagAW3Param.diDecInMS);
	p_NtParamMagAW3AutoSpd				:= ADR(tyNtParamCurr.tyMagAW3Param.diAutoSpdInUMPS);
	p_NtParamMagAW3Tuning				:= ADR(tyNtParamCurr.tyMagAW3Tuning);
	p_NtParamMagAW3EngageSpdInUMPS		:= ADR(tyNtParamCurr.diMagAW3EngageSpdInUMPS);
	p_NtParamMagAW3MotorType			:= ADR(tyNtParamCurr.eMagAW3ServoMotorType);
	p_NtParamMag3WidthOffset			:= ADR(tyNtParamCurr.diMag3WidthOffsetInUM);

	p_NtParamMcProgNm					:= ADR(tyNtParamCurr.sMachineProgNm);

	p_NtParamUSSOT1ProgNm				:= ADR(tyNtParamCurr.sUSSOT1ProgNm);
	p_NtParamUSSOT1RstDlyTm				:= ADR(tyNtParamCurr.tUSSOT1RstDlyTm);
	p_NtParamUSSOT1SigInChkTm			:= ADR(tyNtParamCurr.tUSSOT1SigInChkTm);

	p_NtParamUSSOT2ProgNm				:= ADR(tyNtParamCurr.sUSSOT2ProgNm);
	p_NtParamUSSOT2RstDlyTm				:= ADR(tyNtParamCurr.tUSSOT2RstDlyTm);
	p_NtParamUSSOT2SigInChkTm			:= ADR(tyNtParamCurr.tUSSOT2SigInChkTm);

	p_NtParamUSSOT3ProgNm				:= ADR(tyNtParamCurr.sUSSOT3ProgNm);
	p_NtParamUSSOT3RstDlyTm				:= ADR(tyNtParamCurr.tUSSOT3RstDlyTm);
	p_NtParamUSSOT3SigInChkTm			:= ADR(tyNtParamCurr.tUSSOT3SigInChkTm);

	p_NtParamDSSOT1ProgNm				:= ADR(tyNtParamCurr.sDSSOT1ProgNm);
	p_NtParamDSSOT1RstDlyTm				:= ADR(tyNtParamCurr.tDSSOT1RstDlyTm);
	p_NtParamDSSOT1SigInChkTm			:= ADR(tyNtParamCurr.tDSSOT1SigInChkTm);

	p_NtParamDSSOT2ProgNm				:= ADR(tyNtParamCurr.sDSSOT2ProgNm);
	p_NtParamDSSOT2RstDlyTm				:= ADR(tyNtParamCurr.tDSSOT2RstDlyTm);
	p_NtParamDSSOT2SigInChkTm			:= ADR(tyNtParamCurr.tDSSOT2SigInChkTm);

	p_NtParamDSSOT3ProgNm				:= ADR(tyNtParamCurr.sDSSOT3ProgNm);
	p_NtParamDSSOT3RstDlyTm				:= ADR(tyNtParamCurr.tDSSOT3RstDlyTm);
	p_NtParamDSSOT3SigInChkTm			:= ADR(tyNtParamCurr.tDSSOT3SigInChkTm);

	p_NtParamProjSOTSenPrep				:= ADR(tyNtParamCurr.bProjSOTSensorPrep);
	p_NtParamSOTReadyOnFirst			:= ADR(tyNtParamCurr.bSOTReadyOnFirst);

	p_NtParamShowMESName				:= ADR(tyNtParamCurr.bShowMESName);
	p_NtParamShowFMorMESActive			:= ADR(tyNtParamCurr.bShowFMorMESActive);

	p_NtParamProjUsFixToFixRail			:= ADR(tyNtParamCurr.bProjUSFixToFixRail);
	p_NtParamUIConvDirRL				:= ADR(tyNtParamCurr.bUIConvDirRL);

	p_NtParamProjServoPullPusherPrep	:= ADR(tyNtParamCurr.bProjServoPullerPusherPrep);
	p_NtParamPPProgNm					:= ADR(tyNtParamCurr.sPPProgNm);
	p_NtParamPPDevice					:= ADR(tyNtParamCurr.sPPDevice);
	p_NtParamPPNode						:= ADR(tyNtParamCurr.usiPPNode);
	p_NtParamPPDir						:= ADR(tyNtParamCurr.bPPDir);
	p_NtParamPPDirBl					:= ADR(tyNtParamCurr.bPPDirBl);
	p_NtParamPPPitchInUM				:= ADR(tyNtParamCurr.diPPPitchInUM);
	p_NtParamPPMovBlDistInUM			:= ADR(tyNtParamCurr.diPPMovBlDistInUM);
	p_NtParamPPParamInHm				:= ADR(tyNtParamCurr.tyPPParamInHm);
	p_NtParamPPParamInConvert			:= ADR(tyNtParamCurr.tyPPParamInConvert);
	p_NtParamPPParam					:= ADR(tyNtParamCurr.tyPPParam);
	p_NtParamPPAcc						:= ADR(tyNtParamCurr.tyPPParam.diAccInMS);
	p_NtParamPPDec						:= ADR(tyNtParamCurr.tyPPParam.diDecInMS);
	p_NtParamPPAutoSpd					:= ADR(tyNtParamCurr.tyPPParam.diAutoSpdInUMPS);
	p_NtParamPPTuning					:= ADR(tyNtParamCurr.tyPPTuning);
	p_NtParamPPMotorType				:= ADR(tyNtParamCurr.ePPServoMotorType);

	p_NtParamCurtainSenPrep				:= ADR(tyNtParamCurr.bCurtainSenPrep);
	p_NtParamProjMagHeightChkPrep		:= ADR(tyNtParamCurr.bProjMagHeightChkPrep);
	p_NtParamTravGotoMagWidthChkPt1		:= ADR(tyNtParamCurr.diTravGoToMagWidthChkPt1);
	p_NtParamTravGotoMagWidthChkPt2		:= ADR(tyNtParamCurr.diTravGoToMagWidthChkPt2);
	p_NtParamTravGotoMagWidthChkPt3		:= ADR(tyNtParamCurr.diTravGoToMagWidthChkPt3);

	p_NtParamProjScanPrep				:= ADR(tyNtParamCurr.bProjScanPrep); //Top Btm TCP
	p_NtParamProjOpConPrep				:= ADR(tyNtParamCurr.bProjOpConPrep);
	p_NtParamPPTorqParam				:= ADR(tyNtParamCurr.tyPPTorqParam);
	p_NtParamProjLifTravMnlLoad			:= ADR(tyNtParamCurr.bProjLifTravMnlLoad);

	p_NtParamMidSenNcNo					:= ADR(tyNtParamCurr.eMidSenNcNoType);
	p_NtParamCustomerReq				:=ADR(tyNtParamCurr.eCustomerReq);

	p_NtParamHermesSvyPrep			:= ADR(tyNtParamCurr.bHermesSvyPrep);
	p_NtParamHermesSvyFirstMc		:= ADR(tyNtParamCurr.bHermesSvyFirstMcInTheLine);//First Machine in the line, set for Loader / Destacker
	p_NtParamHermesSvyMagTypeMc		:= ADR(tyNtParamCurr.bHermesSvyMagTypeMc);//Magazine type Machine
	p_NtParamSvyHermesProgNm		:= ADR(tyNtParamCurr.sSvyHermesProgNm);
	p_NtParamSvyHermesConfigFileNm	:= ADR(tyNtParamCurr.sSvyHermesConfigFileNm);
	p_NtParamSvyHermesFileKeepDay	:= ADR(tyNtParamCurr.udiSvyHermesFileKeepDay);
	p_NtParamSvyHermesAliveTmInSec	:= ADR(tyNtParamCurr.udiSvyHermesAliveTmInSec);
	p_NtParamSvyHermesConnTO		:= ADR(tyNtParamCurr.tSvyHermesConnTO);
	p_NtParamSvyHermesRetainFileNm	:= ADR(tyNtParamCurr.sSvyHermesRetainFileNm);
	p_NtParamDSHermesRetainFileNm	:= ADR(tyNtParamCurr.sDSHermesRetainFileNm); //50 Board Data retain file name
	p_NtParamDSHermesMcCycleTm	    := ADR(tyNtParamCurr.rMachineCycleTime); //Machine Board Transfer Cycle Time
	p_NtParamDSHermesAWCycleTm	    := ADR(tyNtParamCurr.rAutoWidthCycleTime); //Machine Autowidth Cycle Time
	p_NtParamHermesScannerPrep    	:= ADR(tyNtParamCurr.bHermesScannerPrep);
	p_NtParamHermesInput            := ADR(tyNtParamCurr.iInput);//Total Input = How many inlet
	p_NtParamHermesOutput           := ADR(tyNtParamCurr.iOutput);//Total Outlet  = How many outlet
	//AutoRcp
	p_NtParamAutoRcpPrep			:= ADR(tyNtParamCurr.bAutoRcpPrep);
	p_NtParamAutoRcpParamLmt		:= ADR(tyNtParamCurr.eAutoRcpParamLmt);
	p_NtParamAutoRcpPrecededBy		:= ADR(tyNtParamCurr.eAutoRcpPrecededBy);
	p_NtParamAutoRcpProgNm			:= ADR(tyNtParamCurr.sAutoRcpProgNm);

	(* Always Change If Project Change *)
	//Inlet Stopper
	p_NtParamProjInletStopperPrep			:= ADR(tyNtParamCurr.bProjInletStopperPrep);
	p_NtParamInletStopperProgNm				:= ADR(tyNtParamCurr.sInletStopperProgNm);
	p_NtParamInletStopperTwoCtrlIn			:= ADR(tyNtParamCurr.bInletStopperTwoCtrlIn);
	p_NtParamInletStopperExtDlyTm			:= ADR(tyNtParamCurr.tInletStopperExtDlyTm);
	p_NtParamInletStopperRetDlyTm			:= ADR(tyNtParamCurr.tInletStopperRetDlyTm);

	//Language
	p_NtParamProjChinesePrep 	:= ADR(tyNtParamCurr.bChinesePrep);
	p_NtParamProjGermanPrep 	:= ADR(tyNtParamCurr.bGermanPrep);

	//HMI Mac Address
	p_NtParamHWInfoHMIMacAddress		:= ADR(tyNtParamCurr.sHWInfoHMIMacAddress);

	p_NtParamAutoRcpF1ArbitraryType		:= ADR(tyNtParamCurr.bAutoRcpF1ArbitratryType);
END_PROGRAM
```

### UsrMgmt.typ - Do Not Change!!!
```iecst
(*2019-05-04*)
(**)
(*Action*)

TYPE
	eUsrMgmtAction :
		(
		UsrMgmtActIdle,
		UsrMgmtActCreateDir,
		UsrMgmtActLogin,
		UsrMgmtActBypassLogin,
		UsrMgmtActLogout,
		UsrMgmtActAdd,
		UsrMgmtActEdit,
		UsrMgmtActDel,
		UsrMgmtActSaveAccessRight,
		UsrMgmtActReadData
		);
END_TYPE

(**)
(*Data*)

TYPE
	tyUsrMgmtParam : 	STRUCT
		sUsrNm : STRING[30];
		sPw : STRING[30];
		eUsrLvl : eUsrMgmtAutLvl;
	END_STRUCT;
	eUsrMgmtAutLvl :
		(
		UsrMgmtLvl1,
		UsrMgmtLvl2,
		UsrMgmtLvl3,
		UsrMgmtAdmin,
		UsrMgmtNtEngr,
		UsrMgmtNtAdmin
		);
	tyUsrMgmtAccessRight : 	STRUCT
		bOpt : BOOL;
		bProdSel : BOOL;
		bMagSel : BOOL;
		bMcInfo : BOOL;
		bAlm : BOOL;
		bBffrInfo : BOOL;
		bOvenInfo : BOOL;
		bMagInfo : BOOL;
		bLFCtrl : BOOL;
		bManual : BOOL;
		bSimulation : BOOL;
		bProdSet : BOOL;
		bMagSet : BOOL;
		bMcSet : BOOL;
		bLang : BOOL;
		bUsrMgmt : BOOL;
		bLFSet : BOOL;
		bChgParam : BOOL;
		bManualFBOnly : BOOL;
		sNm : STRING[30];
	END_STRUCT;
	tyUsrMgmtFullDat : 	STRUCT
		a_tyAllList : ARRAY[1..c_udiUsrMgmtMax]OF tyUsrMgmtParam;
		tyAccessRightLvl1 : tyUsrMgmtAccessRight := (bOpt:=TRUE,bProdSel:=TRUE,bMcInfo:=TRUE,bAlm:=TRUE,bBffrInfo:=TRUE,bOvenInfo:=TRUE,bMagInfo:=TRUE);
		tyAccessRightLvl2 : tyUsrMgmtAccessRight := (bOpt:=TRUE,bProdSel:=TRUE,bMagSel:=TRUE,bMcInfo:=TRUE,bAlm:=TRUE,bBffrInfo:=TRUE,bOvenInfo:=TRUE,bMagInfo:=TRUE,bProdSet:=TRUE,bChgParam:=TRUE,sNm:='Line Leader');
		tyAccessRightLvl3 : tyUsrMgmtAccessRight := (bOpt:=TRUE,bProdSel:=TRUE,bMagSel:=TRUE,bMcInfo:=TRUE,bAlm:=TRUE,bBffrInfo:=TRUE,bOvenInfo:=TRUE,bMagInfo:=TRUE,bLFCtrl:=TRUE,bManual:=TRUE,bSimulation:=TRUE,bProdSet:=TRUE,bMagSet:=TRUE,bMcSet:=TRUE,bLang:=TRUE,bLFSet:=TRUE,bChgParam:=TRUE,sNm:='Technician');
	END_STRUCT;
END_TYPE
```

### Program Logical/UsrMgmt/UsrMgmt (IEC) - 1.00.0 - NtRecipe v5.00.0 , NtFileIO v5.00.0
